	VAR robtarget OpenholeUD_6159 := [[399.17, -20.7, 180.93], [-0.152365, 0.690496, 0.688111, 0.1628], [0,0,0,0], [9E9, 9E9, 9E9, 9E9, 9E9, 9E9]];
	VAR robtarget OpenholeUD_6160 := [[395.17, -20.7, 180.87], [-0.163095, 0.688041, 0.685559, 0.173233], [0,0,0,0], [9E9, 9E9, 9E9, 9E9, 9E9, 9E9]];
	VAR robtarget OpenholeUD_6161 := [[389.34, -20.7, 180.77], [-0.17806, 0.684321, 0.681719, 0.187774], [0,0,0,0], [9E9, 9E9, 9E9, 9E9, 9E9, 9E9]];
	VAR robtarget OpenholeUD_6162 := [[385.34, -20.7, 180.79], [-0.183051, 0.683002, 0.683002, 0.183051], [0,0,0,0], [9E9, 9E9, 9E9, 9E9, 9E9, 9E9]];
	VAR robtarget OpenholeUD_6163 := [[381.34, -20.7, 180.8], [-0.183051, 0.683002, 0.683002, 0.183051], [0,0,0,0], [9E9, 9E9, 9E9, 9E9, 9E9, 9E9]];
	VAR robtarget OpenholeUD_6164 := [[377.34, -20.7, 180.81], [-0.183051, 0.683002, 0.683002, 0.183051], [0,0,0,0], [9E9, 9E9, 9E9, 9E9, 9E9, 9E9]];
	VAR robtarget OpenholeUD_6165 := [[373.34, -20.7, 180.83], [-0.183051, 0.683002, 0.683002, 0.183051], [0,0,0,0], [9E9, 9E9, 9E9, 9E9, 9E9, 9E9]];
	VAR robtarget OpenholeUD_6166 := [[369.34, -20.7, 180.84], [-0.183051, 0.683002, 0.683002, 0.183051], [0,0,0,0], [9E9, 9E9, 9E9, 9E9, 9E9, 9E9]];
	VAR robtarget OpenholeUD_6167 := [[369.34, -20.7, 180.84], [-0.183051, 0.683002, 0.683002, 0.183051], [0,0,0,0], [9E9, 9E9, 9E9, 9E9, 9E9, 9E9]];
	VAR robtarget OpenholeUD_6168 := [[369.35, -19.5, 181.53], [-0.183051, 0.683002, 0.683002, 0.183051], [0,0,0,0], [9E9, 9E9, 9E9, 9E9, 9E9, 9E9]];
	VAR robtarget OpenholeUD_6169 := [[373.35, -19.5, 181.52], [-0.183051, 0.683002, 0.683002, 0.183051], [0,0,0,0], [9E9, 9E9, 9E9, 9E9, 9E9, 9E9]];
	VAR robtarget OpenholeUD_6170 := [[377.35, -19.5, 181.51], [-0.183051, 0.683002, 0.683002, 0.183051], [0,0,0,0], [9E9, 9E9, 9E9, 9E9, 9E9, 9E9]];
	VAR robtarget OpenholeUD_6171 := [[381.35, -19.5, 181.49], [-0.183051, 0.683002, 0.683002, 0.183051], [0,0,0,0], [9E9, 9E9, 9E9, 9E9, 9E9, 9E9]];
	VAR robtarget OpenholeUD_6172 := [[385.35, -19.5, 181.48], [-0.183051, 0.683002, 0.683002, 0.183051], [0,0,0,0], [9E9, 9E9, 9E9, 9E9, 9E9, 9E9]];
	VAR robtarget OpenholeUD_6173 := [[389.35, -19.5, 181.47], [-0.18149, 0.683419, 0.682647, 0.18437], [0,0,0,0], [9E9, 9E9, 9E9, 9E9, 9E9, 9E9]];
	VAR robtarget OpenholeUD_6174 := [[393.35, -19.5, 181.49], [-0.171367, 0.686027, 0.685263, 0.174397], [0,0,0,0], [9E9, 9E9, 9E9, 9E9, 9E9, 9E9]];
	VAR robtarget OpenholeUD_6175 := [[397.35, -19.5, 181.5], [-0.160873, 0.688564, 0.687811, 0.164061], [0,0,0,0], [9E9, 9E9, 9E9, 9E9, 9E9, 9E9]];
	VAR robtarget OpenholeUD_6176 := [[401.35, -19.5, 181.52], [-0.15001, 0.691012, 0.690275, 0.153365], [0,0,0,0], [9E9, 9E9, 9E9, 9E9, 9E9, 9E9]];
	VAR robtarget OpenholeUD_6177 := [[405.35, -19.5, 181.54], [-0.138785, 0.693353, 0.692638, 0.142312], [0,0,0,0], [9E9, 9E9, 9E9, 9E9, 9E9, 9E9]];
	VAR robtarget OpenholeUD_6178 := [[409.35, -19.5, 181.56], [-0.127207, 0.695571, 0.694883, 0.130913], [0,0,0,0], [9E9, 9E9, 9E9, 9E9, 9E9, 9E9]];
	VAR robtarget OpenholeUD_6179 := [[413.35, -19.5, 181.58], [-0.11529, 0.697645, 0.696991, 0.11918], [0,0,0,0], [9E9, 9E9, 9E9, 9E9, 9E9, 9E9]];
	VAR robtarget OpenholeUD_6180 := [[417.35, -19.5, 181.6], [-0.103051, 0.699557, 0.698945, 0.107128], [0,0,0,0], [9E9, 9E9, 9E9, 9E9, 9E9, 9E9]];
	VAR robtarget OpenholeUD_6181 := [[421.35, -19.5, 181.61], [-0.090514, 0.70129, 0.700726, 0.09478], [0,0,0,0], [9E9, 9E9, 9E9, 9E9, 9E9, 9E9]];
	VAR robtarget OpenholeUD_6182 := [[425.35, -19.5, 181.63], [-0.077704, 0.702824, 0.702318, 0.082159], [0,0,0,0], [9E9, 9E9, 9E9, 9E9, 9E9, 9E9]];
	VAR robtarget OpenholeUD_6183 := [[429.35, -19.5, 181.65], [-0.064653, 0.704145, 0.703703, 0.069293], [0,0,0,0], [9E9, 9E9, 9E9, 9E9, 9E9, 9E9]];
	VAR robtarget OpenholeUD_6184 := [[433.35, -19.5, 181.67], [-0.051395, 0.705237, 0.704869, 0.056216], [0,0,0,0], [9E9, 9E9, 9E9, 9E9, 9E9, 9E9]];
	VAR robtarget OpenholeUD_6185 := [[437.35, -19.5, 181.69], [-0.037969, 0.706087, 0.7058, 0.042964], [0,0,0,0], [9E9, 9E9, 9E9, 9E9, 9E9, 9E9]];
	VAR robtarget OpenholeUD_6186 := [[442.9, -19.5, 181.71], [-0.019136, 0.706848, 0.706687, 0.024355], [0,0,0,0], [9E9, 9E9, 9E9, 9E9, 9E9, 9E9]];
	VAR robtarget OpenholeUD_6187 := [[442.9, -19.5, 181.71], [-0.019136, 0.706848, 0.706687, 0.024355], [0,0,0,0], [9E9, 9E9, 9E9, 9E9, 9E9, 9E9]];
	VAR robtarget OpenholeUD_6188 := [[442.86, -18.3, 181.79], [-0.023356, 0.706721, 0.706812, 0.020425], [0,0,0,0], [9E9, 9E9, 9E9, 9E9, 9E9, 9E9]];
	VAR robtarget OpenholeUD_6189 := [[438.86, -18.3, 181.81], [-0.03693, 0.706142, 0.706295, 0.033871], [0,0,0,0], [9E9, 9E9, 9E9, 9E9, 9E9, 9E9]];
	VAR robtarget OpenholeUD_6190 := [[434.86, -18.3, 181.84], [-0.050386, 0.705309, 0.705529, 0.047203], [0,0,0,0], [9E9, 9E9, 9E9, 9E9, 9E9, 9E9]];
	VAR robtarget OpenholeUD_6191 := [[430.86, -18.3, 181.87], [-0.063682, 0.704233, 0.704524, 0.06038], [0,0,0,0], [9E9, 9E9, 9E9, 9E9, 9E9, 9E9]];
	VAR robtarget OpenholeUD_6192 := [[426.86, -18.3, 181.9], [-0.076779, 0.702926, 0.70329, 0.073366], [0,0,0,0], [9E9, 9E9, 9E9, 9E9, 9E9, 9E9]];
	VAR robtarget OpenholeUD_6193 := [[422.86, -18.3, 181.93], [-0.089642, 0.701402, 0.701842, 0.086125], [0,0,0,0], [9E9, 9E9, 9E9, 9E9, 9E9, 9E9]];
	VAR robtarget OpenholeUD_6194 := [[418.86, -18.3, 181.95], [-0.102237, 0.699677, 0.700195, 0.098627], [0,0,0,0], [9E9, 9E9, 9E9, 9E9, 9E9, 9E9]];
	VAR robtarget OpenholeUD_6195 := [[414.86, -18.3, 181.98], [-0.114539, 0.697769, 0.698365, 0.110845], [0,0,0,0], [9E9, 9E9, 9E9, 9E9, 9E9, 9E9]];
	VAR robtarget OpenholeUD_6196 := [[410.86, -18.3, 182.01], [-0.126522, 0.695695, 0.69637, 0.122757], [0,0,0,0], [9E9, 9E9, 9E9, 9E9, 9E9, 9E9]];
	VAR robtarget OpenholeUD_6197 := [[406.86, -18.3, 182.04], [-0.138169, 0.693476, 0.694227, 0.134344], [0,0,0,0], [9E9, 9E9, 9E9, 9E9, 9E9, 9E9]];
	VAR robtarget OpenholeUD_6198 := [[402.86, -18.3, 182.07], [-0.149465, 0.69113, 0.691956, 0.145591], [0,0,0,0], [9E9, 9E9, 9E9, 9E9, 9E9, 9E9]];
	VAR robtarget OpenholeUD_6199 := [[398.86, -18.3, 182.09], [-0.160399, 0.688674, 0.689573, 0.156488], [0,0,0,0], [9E9, 9E9, 9E9, 9E9, 9E9, 9E9]];
	VAR robtarget OpenholeUD_6200 := [[394.86, -18.3, 182.12], [-0.170965, 0.686128, 0.687096, 0.167028], [0,0,0,0], [9E9, 9E9, 9E9, 9E9, 9E9, 9E9]];
	VAR robtarget OpenholeUD_6201 := [[389.35, -18.3, 182.16], [-0.184916, 0.6825, 0.683559, 0.180962], [0,0,0,0], [9E9, 9E9, 9E9, 9E9, 9E9, 9E9]];
	VAR robtarget OpenholeUD_6202 := [[385.35, -18.3, 182.17], [-0.183051, 0.683002, 0.683002, 0.183051], [0,0,0,0], [9E9, 9E9, 9E9, 9E9, 9E9, 9E9]];
	VAR robtarget OpenholeUD_6203 := [[381.35, -18.3, 182.19], [-0.183051, 0.683002, 0.683002, 0.183051], [0,0,0,0], [9E9, 9E9, 9E9, 9E9, 9E9, 9E9]];
	VAR robtarget OpenholeUD_6204 := [[377.35, -18.3, 182.2], [-0.183051, 0.683002, 0.683002, 0.183051], [0,0,0,0], [9E9, 9E9, 9E9, 9E9, 9E9, 9E9]];
	VAR robtarget OpenholeUD_6205 := [[373.35, -18.3, 182.21], [-0.183051, 0.683002, 0.683002, 0.183051], [0,0,0,0], [9E9, 9E9, 9E9, 9E9, 9E9, 9E9]];
	VAR robtarget OpenholeUD_6206 := [[369.35, -18.3, 182.22], [-0.183051, 0.683002, 0.683002, 0.183051], [0,0,0,0], [9E9, 9E9, 9E9, 9E9, 9E9, 9E9]];
	VAR robtarget OpenholeUD_6207 := [[369.35, -18.3, 182.22], [-0.183051, 0.683002, 0.683002, 0.183051], [0,0,0,0], [9E9, 9E9, 9E9, 9E9, 9E9, 9E9]];
	VAR robtarget OpenholeUD_6208 := [[369.35, -17.1, 182.92], [-0.183051, 0.683002, 0.683002, 0.183051], [0,0,0,0], [9E9, 9E9, 9E9, 9E9, 9E9, 9E9]];
	VAR robtarget OpenholeUD_6209 := [[373.35, -17.1, 182.9], [-0.183051, 0.683002, 0.683002, 0.183051], [0,0,0,0], [9E9, 9E9, 9E9, 9E9, 9E9, 9E9]];
	VAR robtarget OpenholeUD_6210 := [[377.35, -17.1, 182.89], [-0.183051, 0.683002, 0.683002, 0.183051], [0,0,0,0], [9E9, 9E9, 9E9, 9E9, 9E9, 9E9]];
	VAR robtarget OpenholeUD_6211 := [[381.35, -17.1, 182.88], [-0.183051, 0.683002, 0.683002, 0.183051], [0,0,0,0], [9E9, 9E9, 9E9, 9E9, 9E9, 9E9]];
	VAR robtarget OpenholeUD_6212 := [[389.35, -17.1, 182.85], [-0.188337, 0.681564, 0.684453, 0.17755], [0,0,0,0], [9E9, 9E9, 9E9, 9E9, 9E9, 9E9]];
	VAR robtarget OpenholeUD_6213 := [[393.35, -17.1, 182.78], [-0.178356, 0.684243, 0.686996, 0.167441], [0,0,0,0], [9E9, 9E9, 9E9, 9E9, 9E9, 9E9]];
	VAR robtarget OpenholeUD_6214 := [[397.35, -17.1, 182.71], [-0.168002, 0.686859, 0.689464, 0.156971], [0,0,0,0], [9E9, 9E9, 9E9, 9E9, 9E9, 9E9]];
	VAR robtarget OpenholeUD_6215 := [[401.35, -17.1, 182.63], [-0.157276, 0.689394, 0.69184, 0.146144], [0,0,0,0], [9E9, 9E9, 9E9, 9E9, 9E9, 9E9]];
	VAR robtarget OpenholeUD_6216 := [[405.35, -17.1, 182.56], [-0.146183, 0.691831, 0.694107, 0.134966], [0,0,0,0], [9E9, 9E9, 9E9, 9E9, 9E9, 9E9]];
	VAR robtarget OpenholeUD_6217 := [[409.35, -17.1, 182.48], [-0.134731, 0.694152, 0.696248, 0.123447], [0,0,0,0], [9E9, 9E9, 9E9, 9E9, 9E9, 9E9]];
	VAR robtarget OpenholeUD_6218 := [[413.35, -17.1, 182.41], [-0.122934, 0.696338, 0.698244, 0.111601], [0,0,0,0], [9E9, 9E9, 9E9, 9E9, 9E9, 9E9]];
	VAR robtarget OpenholeUD_6219 := [[417.35, -17.1, 182.33], [-0.110807, 0.698371, 0.700079, 0.099445], [0,0,0,0], [9E9, 9E9, 9E9, 9E9, 9E9, 9E9]];
	VAR robtarget OpenholeUD_6220 := [[421.35, -17.1, 182.26], [-0.098372, 0.700231, 0.701734, 0.087], [0,0,0,0], [9E9, 9E9, 9E9, 9E9, 9E9, 9E9]];
	VAR robtarget OpenholeUD_6221 := [[425.34, -17.1, 182.19], [-0.085654, 0.7019, 0.703193, 0.074294], [0,0,0,0], [9E9, 9E9, 9E9, 9E9, 9E9, 9E9]];
	VAR robtarget OpenholeUD_6222 := [[429.34, -17.1, 182.11], [-0.072683, 0.703361, 0.70444, 0.061354], [0,0,0,0], [9E9, 9E9, 9E9, 9E9, 9E9, 9E9]];
	VAR robtarget OpenholeUD_6223 := [[433.34, -17.1, 182.04], [-0.059492, 0.7046, 0.705461, 0.048215], [0,0,0,0], [9E9, 9E9, 9E9, 9E9, 9E9, 9E9]];
	VAR robtarget OpenholeUD_6224 := [[437.34, -17.1, 181.96], [-0.04612, 0.705601, 0.706244, 0.034914], [0,0,0,0], [9E9, 9E9, 9E9, 9E9, 9E9, 9E9]];
	VAR robtarget OpenholeUD_6225 := [[443.05, -17.1, 181.86], [-0.02681, 0.706598, 0.706932, 0.015737], [0,0,0,0], [9E9, 9E9, 9E9, 9E9, 9E9, 9E9]];
	VAR robtarget OpenholeUD_6226 := [[443.05, -17.1, 181.86], [-0.02681, 0.706598, 0.706932, 0.015737], [0,0,0,0], [9E9, 9E9, 9E9, 9E9, 9E9, 9E9]];
	VAR robtarget OpenholeUD_6227 := [[443.48, -15.9, 181.92], [-0.029424, 0.706494, 0.707033, 0.010217], [0,0,0,0], [9E9, 9E9, 9E9, 9E9, 9E9, 9E9]];
	VAR robtarget OpenholeUD_6228 := [[439.48, -15.9, 182.04], [-0.042977, 0.7058, 0.70671, 0.023699], [0,0,0,0], [9E9, 9E9, 9E9, 9E9, 9E9, 9E9]];
	VAR robtarget OpenholeUD_6229 := [[435.49, -15.9, 182.16], [-0.056403, 0.704854, 0.706133, 0.037088], [0,0,0,0], [9E9, 9E9, 9E9, 9E9, 9E9, 9E9]];
	VAR robtarget OpenholeUD_6230 := [[431.49, -15.9, 182.28], [-0.069663, 0.703667, 0.705312, 0.050343], [0,0,0,0], [9E9, 9E9, 9E9, 9E9, 9E9, 9E9]];
	VAR robtarget OpenholeUD_6231 := [[427.49, -15.9, 182.4], [-0.082716, 0.702252, 0.704257, 0.063424], [0,0,0,0], [9E9, 9E9, 9E9, 9E9, 9E9, 9E9]];
	VAR robtarget OpenholeUD_6232 := [[423.49, -15.9, 182.52], [-0.095528, 0.700624, 0.702979, 0.076296], [0,0,0,0], [9E9, 9E9, 9E9, 9E9, 9E9, 9E9]];
	VAR robtarget OpenholeUD_6233 := [[419.49, -15.9, 182.64], [-0.108067, 0.6988, 0.701493, 0.088927], [0,0,0,0], [9E9, 9E9, 9E9, 9E9, 9E9, 9E9]];
	VAR robtarget OpenholeUD_6234 := [[415.49, -15.9, 182.76], [-0.120306, 0.696797, 0.699815, 0.101288], [0,0,0,0], [9E9, 9E9, 9E9, 9E9, 9E9, 9E9]];
	VAR robtarget OpenholeUD_6235 := [[411.5, -15.9, 182.88], [-0.132222, 0.694635, 0.697962, 0.113355], [0,0,0,0], [9E9, 9E9, 9E9, 9E9, 9E9, 9E9]];
	VAR robtarget OpenholeUD_6236 := [[407.5, -15.9, 183], [-0.143797, 0.692331, 0.695951, 0.125107], [0,0,0,0], [9E9, 9E9, 9E9, 9E9, 9E9, 9E9]];
	VAR robtarget OpenholeUD_6237 := [[403.5, -15.9, 183.12], [-0.155017, 0.689906, 0.693801, 0.136528], [0,0,0,0], [9E9, 9E9, 9E9, 9E9, 9E9, 9E9]];
	VAR robtarget OpenholeUD_6238 := [[399.5, -15.9, 183.24], [-0.165872, 0.687377, 0.691529, 0.147606], [0,0,0,0], [9E9, 9E9, 9E9, 9E9, 9E9, 9E9]];
	VAR robtarget OpenholeUD_6239 := [[395.5, -15.9, 183.36], [-0.176355, 0.684762, 0.689152, 0.158332], [0,0,0,0], [9E9, 9E9, 9E9, 9E9, 9E9, 9E9]];
	VAR robtarget OpenholeUD_6240 := [[389.35, -15.9, 183.55], [-0.191751, 0.680611, 0.68533, 0.174134], [0,0,0,0], [9E9, 9E9, 9E9, 9E9, 9E9, 9E9]];
	VAR robtarget OpenholeUD_6241 := [[385.35, -15.9, 183.56], [-0.183051, 0.683002, 0.683002, 0.183051], [0,0,0,0], [9E9, 9E9, 9E9, 9E9, 9E9, 9E9]];
	VAR robtarget OpenholeUD_6242 := [[381.35, -15.9, 183.57], [-0.183051, 0.683002, 0.683002, 0.183051], [0,0,0,0], [9E9, 9E9, 9E9, 9E9, 9E9, 9E9]];
	VAR robtarget OpenholeUD_6243 := [[377.35, -15.9, 183.58], [-0.183051, 0.683002, 0.683002, 0.183051], [0,0,0,0], [9E9, 9E9, 9E9, 9E9, 9E9, 9E9]];
	VAR robtarget OpenholeUD_6244 := [[369.35, -15.9, 183.61], [-0.183051, 0.683002, 0.683002, 0.183051], [0,0,0,0], [9E9, 9E9, 9E9, 9E9, 9E9, 9E9]];
	VAR robtarget OpenholeUD_6245 := [[369.35, -15.9, 183.61], [-0.183051, 0.683002, 0.683002, 0.183051], [0,0,0,0], [9E9, 9E9, 9E9, 9E9, 9E9, 9E9]];
	VAR robtarget OpenholeUD_6246 := [[369.36, -14.7, 184.3], [-0.183051, 0.683002, 0.683002, 0.183051], [0,0,0,0], [9E9, 9E9, 9E9, 9E9, 9E9, 9E9]];
	VAR robtarget OpenholeUD_6247 := [[373.36, -14.7, 184.29], [-0.183051, 0.683002, 0.683002, 0.183051], [0,0,0,0], [9E9, 9E9, 9E9, 9E9, 9E9, 9E9]];
	VAR robtarget OpenholeUD_6248 := [[377.36, -14.7, 184.28], [-0.183051, 0.683002, 0.683002, 0.183051], [0,0,0,0], [9E9, 9E9, 9E9, 9E9, 9E9, 9E9]];
	VAR robtarget OpenholeUD_6249 := [[381.36, -14.7, 184.27], [-0.183051, 0.683002, 0.683002, 0.183051], [0,0,0,0], [9E9, 9E9, 9E9, 9E9, 9E9, 9E9]];
	VAR robtarget OpenholeUD_6250 := [[389.36, -14.7, 184.24], [-0.195159, 0.679642, 0.686189, 0.170717], [0,0,0,0], [9E9, 9E9, 9E9, 9E9, 9E9, 9E9]];
	VAR robtarget OpenholeUD_6251 := [[393.35, -14.7, 184.07], [-0.185327, 0.682389, 0.688656, 0.160477], [0,0,0,0], [9E9, 9E9, 9E9, 9E9, 9E9, 9E9]];
	VAR robtarget OpenholeUD_6252 := [[397.35, -14.7, 183.91], [-0.175118, 0.685079, 0.69104, 0.149881], [0,0,0,0], [9E9, 9E9, 9E9, 9E9, 9E9, 9E9]];
	VAR robtarget OpenholeUD_6253 := [[401.34, -14.7, 183.74], [-0.164535, 0.687698, 0.693324, 0.138931], [0,0,0,0], [9E9, 9E9, 9E9, 9E9, 9E9, 9E9]];
	VAR robtarget OpenholeUD_6254 := [[405.34, -14.7, 183.57], [-0.153582, 0.690227, 0.695492, 0.127635], [0,0,0,0], [9E9, 9E9, 9E9, 9E9, 9E9, 9E9]];
	VAR robtarget OpenholeUD_6255 := [[409.34, -14.7, 183.41], [-0.142264, 0.692648, 0.697526, 0.116004], [0,0,0,0], [9E9, 9E9, 9E9, 9E9, 9E9, 9E9]];
	VAR robtarget OpenholeUD_6256 := [[413.33, -14.7, 183.24], [-0.130595, 0.694942, 0.699409, 0.104054], [0,0,0,0], [9E9, 9E9, 9E9, 9E9, 9E9, 9E9]];
	VAR robtarget OpenholeUD_6257 := [[417.33, -14.7, 183.07], [-0.118588, 0.697092, 0.701122, 0.091801], [0,0,0,0], [9E9, 9E9, 9E9, 9E9, 9E9, 9E9]];
	VAR robtarget OpenholeUD_6258 := [[421.33, -14.7, 182.91], [-0.106265, 0.699076, 0.702649, 0.079271], [0,0,0,0], [9E9, 9E9, 9E9, 9E9, 9E9, 9E9]];
	VAR robtarget OpenholeUD_6259 := [[425.32, -14.7, 182.74], [-0.093648, 0.700878, 0.703974, 0.066488], [0,0,0,0], [9E9, 9E9, 9E9, 9E9, 9E9, 9E9]];
	VAR robtarget OpenholeUD_6260 := [[429.32, -14.7, 182.58], [-0.080766, 0.702479, 0.705081, 0.053484], [0,0,0,0], [9E9, 9E9, 9E9, 9E9, 9E9, 9E9]];
	VAR robtarget OpenholeUD_6261 := [[433.32, -14.7, 182.41], [-0.067653, 0.703863, 0.705958, 0.040293], [0,0,0,0], [9E9, 9E9, 9E9, 9E9, 9E9, 9E9]];
	VAR robtarget OpenholeUD_6262 := [[437.31, -14.7, 182.24], [-0.054344, 0.705015, 0.706593, 0.026953], [0,0,0,0], [9E9, 9E9, 9E9, 9E9, 9E9, 9E9]];
	VAR robtarget OpenholeUD_6263 := [[444.22, -14.7, 181.95], [-0.030987, 0.706427, 0.707097, 0.003651], [0,0,0,0], [9E9, 9E9, 9E9, 9E9, 9E9, 9E9]];
	VAR robtarget OpenholeUD_6264 := [[444.22, -14.7, 181.95], [-0.030987, 0.706427, 0.707097, 0.003651], [0,0,0,0], [9E9, 9E9, 9E9, 9E9, 9E9, 9E9]];
	VAR robtarget OpenholeUD_6265 := [[445.45, -13.5, 181.95], [-0.030912, 0.706431, 0.707092, -0.004543], [0,0,0,0], [9E9, 9E9, 9E9, 9E9, 9E9, 9E9]];
	VAR robtarget OpenholeUD_6266 := [[441.45, -13.5, 182.16], [-0.044472, 0.705707, 0.70705, 0.008977], [0,0,0,0], [9E9, 9E9, 9E9, 9E9, 9E9, 9E9]];
	VAR robtarget OpenholeUD_6267 := [[437.46, -13.5, 182.37], [-0.057913, 0.704731, 0.706751, 0.022438], [0,0,0,0], [9E9, 9E9, 9E9, 9E9, 9E9, 9E9]];
	VAR robtarget OpenholeUD_6268 := [[433.46, -13.5, 182.59], [-0.071194, 0.703514, 0.7062, 0.0358], [0,0,0,0], [9E9, 9E9, 9E9, 9E9, 9E9, 9E9]];
	VAR robtarget OpenholeUD_6269 := [[429.47, -13.5, 182.8], [-0.084275, 0.702067, 0.705406, 0.04902], [0,0,0,0], [9E9, 9E9, 9E9, 9E9, 9E9, 9E9]];
	VAR robtarget OpenholeUD_6270 := [[425.48, -13.5, 183.01], [-0.097118, 0.700406, 0.704378, 0.062061], [0,0,0,0], [9E9, 9E9, 9E9, 9E9, 9E9, 9E9]];
	VAR robtarget OpenholeUD_6271 := [[421.48, -13.5, 183.22], [-0.109693, 0.698547, 0.70313, 0.074888], [0,0,0,0], [9E9, 9E9, 9E9, 9E9, 9E9, 9E9]];
	VAR robtarget OpenholeUD_6272 := [[417.49, -13.5, 183.44], [-0.121971, 0.696508, 0.701676, 0.08747], [0,0,0,0], [9E9, 9E9, 9E9, 9E9, 9E9, 9E9]];
	VAR robtarget OpenholeUD_6273 := [[413.49, -13.5, 183.65], [-0.133929, 0.694308, 0.700032, 0.099779], [0,0,0,0], [9E9, 9E9, 9E9, 9E9, 9E9, 9E9]];
	VAR robtarget OpenholeUD_6274 := [[409.5, -13.5, 183.86], [-0.145546, 0.691966, 0.698214, 0.111792], [0,0,0,0], [9E9, 9E9, 9E9, 9E9, 9E9, 9E9]];
	VAR robtarget OpenholeUD_6275 := [[405.5, -13.5, 184.07], [-0.156809, 0.6895, 0.69624, 0.123489], [0,0,0,0], [9E9, 9E9, 9E9, 9E9, 9E9, 9E9]];
	VAR robtarget OpenholeUD_6276 := [[401.51, -13.5, 184.29], [-0.167706, 0.686931, 0.694128, 0.134855], [0,0,0,0], [9E9, 9E9, 9E9, 9E9, 9E9, 9E9]];
	VAR robtarget OpenholeUD_6277 := [[397.52, -13.5, 184.5], [-0.178231, 0.684276, 0.691896, 0.145878], [0,0,0,0], [9E9, 9E9, 9E9, 9E9, 9E9, 9E9]];
	VAR robtarget OpenholeUD_6278 := [[393.52, -13.5, 184.71], [-0.18838, 0.681552, 0.689559, 0.156551], [0,0,0,0], [9E9, 9E9, 9E9, 9E9, 9E9, 9E9]];
	VAR robtarget OpenholeUD_6279 := [[389.36, -13.5, 184.93], [-0.19856, 0.678656, 0.687031, 0.167297], [0,0,0,0], [9E9, 9E9, 9E9, 9E9, 9E9, 9E9]];
	VAR robtarget OpenholeUD_6280 := [[385.36, -13.5, 184.95], [-0.183051, 0.683002, 0.683002, 0.183051], [0,0,0,0], [9E9, 9E9, 9E9, 9E9, 9E9, 9E9]];
	VAR robtarget OpenholeUD_6281 := [[381.36, -13.5, 184.96], [-0.183051, 0.683002, 0.683002, 0.183051], [0,0,0,0], [9E9, 9E9, 9E9, 9E9, 9E9, 9E9]];
	VAR robtarget OpenholeUD_6282 := [[377.36, -13.5, 184.97], [-0.183051, 0.683002, 0.683002, 0.183051], [0,0,0,0], [9E9, 9E9, 9E9, 9E9, 9E9, 9E9]];
	VAR robtarget OpenholeUD_6283 := [[369.36, -13.5, 185], [-0.183051, 0.683002, 0.683002, 0.183051], [0,0,0,0], [9E9, 9E9, 9E9, 9E9, 9E9, 9E9]];
	VAR robtarget OpenholeUD_6284 := [[369.36, -13.5, 185], [-0.183051, 0.683002, 0.683002, 0.183051], [0,0,0,0], [9E9, 9E9, 9E9, 9E9, 9E9, 9E9]];
	VAR robtarget OpenholeUD_6285 := [[369.36, -12.3, 185.69], [-0.183051, 0.683002, 0.683002, 0.183051], [0,0,0,0], [9E9, 9E9, 9E9, 9E9, 9E9, 9E9]];
	VAR robtarget OpenholeUD_6286 := [[373.36, -12.3, 185.68], [-0.183051, 0.683002, 0.683002, 0.183051], [0,0,0,0], [9E9, 9E9, 9E9, 9E9, 9E9, 9E9]];
	VAR robtarget OpenholeUD_6287 := [[377.36, -12.3, 185.66], [-0.183051, 0.683002, 0.683002, 0.183051], [0,0,0,0], [9E9, 9E9, 9E9, 9E9, 9E9, 9E9]];
	VAR robtarget OpenholeUD_6288 := [[381.36, -12.3, 185.65], [-0.183051, 0.683002, 0.683002, 0.183051], [0,0,0,0], [9E9, 9E9, 9E9, 9E9, 9E9, 9E9]];
	VAR robtarget OpenholeUD_6289 := [[385.36, -12.3, 185.64], [-0.183051, 0.683002, 0.683002, 0.183051], [0,0,0,0], [9E9, 9E9, 9E9, 9E9, 9E9, 9E9]];
	VAR robtarget OpenholeUD_6290 := [[389.36, -12.3, 185.63], [-0.201952, 0.677654, 0.687855, 0.163877], [0,0,0,0], [9E9, 9E9, 9E9, 9E9, 9E9, 9E9]];
	VAR robtarget OpenholeUD_6291 := [[393.35, -12.3, 185.37], [-0.192272, 0.680464, 0.690241, 0.153515], [0,0,0,0], [9E9, 9E9, 9E9, 9E9, 9E9, 9E9]];
	VAR robtarget OpenholeUD_6292 := [[397.34, -12.3, 185.11], [-0.182215, 0.683226, 0.692538, 0.142798], [0,0,0,0], [9E9, 9E9, 9E9, 9E9, 9E9, 9E9]];
	VAR robtarget OpenholeUD_6293 := [[401.33, -12.3, 184.85], [-0.171781, 0.685924, 0.694728, 0.131733], [0,0,0,0], [9E9, 9E9, 9E9, 9E9, 9E9, 9E9]];
	VAR robtarget OpenholeUD_6294 := [[405.33, -12.3, 184.59], [-0.160973, 0.68854, 0.696794, 0.120328], [0,0,0,0], [9E9, 9E9, 9E9, 9E9, 9E9, 9E9]];
	VAR robtarget OpenholeUD_6295 := [[409.32, -12.3, 184.33], [-0.149797, 0.691058, 0.698718, 0.108594], [0,0,0,0], [9E9, 9E9, 9E9, 9E9, 9E9, 9E9]];
	VAR robtarget OpenholeUD_6296 := [[413.31, -12.3, 184.08], [-0.138263, 0.693458, 0.700485, 0.096548], [0,0,0,0], [9E9, 9E9, 9E9, 9E9, 9E9, 9E9]];
	VAR robtarget OpenholeUD_6297 := [[417.3, -12.3, 183.82], [-0.126385, 0.69572, 0.702075, 0.084208], [0,0,0,0], [9E9, 9E9, 9E9, 9E9, 9E9, 9E9]];
	VAR robtarget OpenholeUD_6298 := [[421.29, -12.3, 183.56], [-0.114181, 0.697827, 0.703472, 0.0716], [0,0,0,0], [9E9, 9E9, 9E9, 9E9, 9E9, 9E9]];
	VAR robtarget OpenholeUD_6299 := [[425.28, -12.3, 183.3], [-0.101674, 0.699759, 0.704662, 0.058751], [0,0,0,0], [9E9, 9E9, 9E9, 9E9, 9E9, 9E9]];
	VAR robtarget OpenholeUD_6300 := [[429.28, -12.3, 183.04], [-0.088892, 0.701497, 0.705629, 0.045692], [0,0,0,0], [9E9, 9E9, 9E9, 9E9, 9E9, 9E9]];
	VAR robtarget OpenholeUD_6301 := [[433.27, -12.3, 182.78], [-0.075866, 0.703025, 0.706361, 0.032458], [0,0,0,0], [9E9, 9E9, 9E9, 9E9, 9E9, 9E9]];
	VAR robtarget OpenholeUD_6302 := [[437.26, -12.3, 182.52], [-0.062631, 0.704328, 0.706849, 0.019088], [0,0,0,0], [9E9, 9E9, 9E9, 9E9, 9E9, 9E9]];
	VAR robtarget OpenholeUD_6303 := [[441.25, -12.3, 182.27], [-0.049226, 0.705391, 0.707084, 0.005623], [0,0,0,0], [9E9, 9E9, 9E9, 9E9, 9E9, 9E9]];
	VAR robtarget OpenholeUD_6304 := [[445.24, -12.3, 182.01], [-0.035693, 0.706205, 0.707063, -0.007895], [0,0,0,0], [9E9, 9E9, 9E9, 9E9, 9E9, 9E9]];
	VAR robtarget OpenholeUD_6305 := [[449.23, -12.3, 181.75], [-0.022077, 0.706762, 0.706782, -0.021422], [0,0,0,0], [9E9, 9E9, 9E9, 9E9, 9E9, 9E9]];
	VAR robtarget OpenholeUD_6306 := [[453.23, -12.3, 181.49], [-0.008423, 0.707057, 0.706244, -0.034914], [0,0,0,0], [9E9, 9E9, 9E9, 9E9, 9E9, 9E9]];
	VAR robtarget OpenholeUD_6307 := [[457.22, -12.3, 181.23], [0.005224, 0.707087, 0.705453, -0.048326], [0,0,0,0], [9E9, 9E9, 9E9, 9E9, 9E9, 9E9]];
	VAR robtarget OpenholeUD_6308 := [[461.21, -12.3, 180.97], [0.018817, 0.706856, 0.704417, -0.061617], [0,0,0,0], [9E9, 9E9, 9E9, 9E9, 9E9, 9E9]];
	VAR robtarget OpenholeUD_6309 := [[465.2, -12.3, 180.71], [0.032313, 0.706368, 0.703145, -0.074746], [0,0,0,0], [9E9, 9E9, 9E9, 9E9, 9E9, 9E9]];
	VAR robtarget OpenholeUD_6310 := [[469.19, -12.3, 180.46], [0.045667, 0.705631, 0.70165, -0.087675], [0,0,0,0], [9E9, 9E9, 9E9, 9E9, 9E9, 9E9]];
	VAR robtarget OpenholeUD_6311 := [[473.18, -12.3, 180.2], [0.058842, 0.704654, 0.699947, -0.10037], [0,0,0,0], [9E9, 9E9, 9E9, 9E9, 9E9, 9E9]];
	VAR robtarget OpenholeUD_6312 := [[477.18, -12.3, 179.94], [0.0718, 0.703452, 0.698052, -0.112799], [0,0,0,0], [9E9, 9E9, 9E9, 9E9, 9E9, 9E9]];
	VAR robtarget OpenholeUD_6313 := [[481.17, -12.3, 179.68], [0.08451, 0.702039, 0.695982, -0.124937], [0,0,0,0], [9E9, 9E9, 9E9, 9E9, 9E9, 9E9]];
	VAR robtarget OpenholeUD_6314 := [[485.16, -12.3, 179.42], [0.096942, 0.70043, 0.693756, -0.13676], [0,0,0,0], [9E9, 9E9, 9E9, 9E9, 9E9, 9E9]];
	VAR robtarget OpenholeUD_6315 := [[489.15, -12.3, 179.16], [0.109072, 0.698644, 0.691391, -0.148249], [0,0,0,0], [9E9, 9E9, 9E9, 9E9, 9E9, 9E9]];
	VAR robtarget OpenholeUD_6316 := [[493.14, -12.3, 178.91], [0.12088, 0.696698, 0.688908, -0.159391], [0,0,0,0], [9E9, 9E9, 9E9, 9E9, 9E9, 9E9]];
	VAR robtarget OpenholeUD_6317 := [[497.13, -12.3, 178.65], [0.132351, 0.69461, 0.686324, -0.170175], [0,0,0,0], [9E9, 9E9, 9E9, 9E9, 9E9, 9E9]];
	VAR robtarget OpenholeUD_6318 := [[501.13, -12.3, 178.39], [0.143473, 0.692398, 0.683656, -0.180593], [0,0,0,0], [9E9, 9E9, 9E9, 9E9, 9E9, 9E9]];
	VAR robtarget OpenholeUD_6319 := [[505.12, -12.3, 178.13], [0.154238, 0.69008, 0.680922, -0.190644], [0,0,0,0], [9E9, 9E9, 9E9, 9E9, 9E9, 9E9]];
	VAR robtarget OpenholeUD_6320 := [[509.34, -12.3, 177.86], [0.183051, 0.683002, 0.683002, -0.183051], [0,0,0,0], [9E9, 9E9, 9E9, 9E9, 9E9, 9E9]];
	VAR robtarget OpenholeUD_6321 := [[513.34, -12.3, 177.84], [0.183051, 0.683002, 0.683002, -0.183051], [0,0,0,0], [9E9, 9E9, 9E9, 9E9, 9E9, 9E9]];
	VAR robtarget OpenholeUD_6322 := [[517.34, -12.3, 177.83], [0.183051, 0.683002, 0.683002, -0.183051], [0,0,0,0], [9E9, 9E9, 9E9, 9E9, 9E9, 9E9]];
	VAR robtarget OpenholeUD_6323 := [[521.34, -12.3, 177.82], [0.183051, 0.683002, 0.683002, -0.183051], [0,0,0,0], [9E9, 9E9, 9E9, 9E9, 9E9, 9E9]];
	VAR robtarget OpenholeUD_6324 := [[529.34, -12.3, 177.79], [0.183051, 0.683002, 0.683002, -0.183051], [0,0,0,0], [9E9, 9E9, 9E9, 9E9, 9E9, 9E9]];
	VAR robtarget OpenholeUD_6325 := [[529.34, -12.3, 177.79], [0.183051, 0.683002, 0.683002, -0.183051], [0,0,0,0], [9E9, 9E9, 9E9, 9E9, 9E9, 9E9]];
	VAR robtarget OpenholeUD_6326 := [[529.34, -13.5, 178.49], [0.183051, 0.683002, 0.683002, -0.183051], [0,0,0,0], [9E9, 9E9, 9E9, 9E9, 9E9, 9E9]];
	VAR robtarget OpenholeUD_6327 := [[525.34, -13.5, 178.5], [0.183051, 0.683002, 0.683002, -0.183051], [0,0,0,0], [9E9, 9E9, 9E9, 9E9, 9E9, 9E9]];
	VAR robtarget OpenholeUD_6328 := [[521.34, -13.5, 178.51], [0.183051, 0.683002, 0.683002, -0.183051], [0,0,0,0], [9E9, 9E9, 9E9, 9E9, 9E9, 9E9]];
	VAR robtarget OpenholeUD_6329 := [[517.34, -13.5, 178.52], [0.183051, 0.683002, 0.683002, -0.183051], [0,0,0,0], [9E9, 9E9, 9E9, 9E9, 9E9, 9E9]];
	VAR robtarget OpenholeUD_6330 := [[513.34, -13.5, 178.54], [0.183051, 0.683002, 0.683002, -0.183051], [0,0,0,0], [9E9, 9E9, 9E9, 9E9, 9E9, 9E9]];
	VAR robtarget OpenholeUD_6331 := [[509.34, -13.5, 178.55], [0.183051, 0.683002, 0.683002, -0.183051], [0,0,0,0], [9E9, 9E9, 9E9, 9E9, 9E9, 9E9]];
	VAR robtarget OpenholeUD_6332 := [[505.34, -13.5, 178.76], [0.158342, 0.68915, 0.681724, -0.187755], [0,0,0,0], [9E9, 9E9, 9E9, 9E9, 9E9, 9E9]];
	VAR robtarget OpenholeUD_6333 := [[501.35, -13.5, 178.97], [0.147659, 0.691518, 0.684427, -0.177651], [0,0,0,0], [9E9, 9E9, 9E9, 9E9, 9E9, 9E9]];
	VAR robtarget OpenholeUD_6334 := [[497.35, -13.5, 179.19], [0.136615, 0.693784, 0.68706, -0.16718], [0,0,0,0], [9E9, 9E9, 9E9, 9E9, 9E9, 9E9]];
	VAR robtarget OpenholeUD_6335 := [[493.36, -13.5, 179.4], [0.125219, 0.695931, 0.689606, -0.156345], [0,0,0,0], [9E9, 9E9, 9E9, 9E9, 9E9, 9E9]];
	VAR robtarget OpenholeUD_6336 := [[489.37, -13.5, 179.61], [0.113482, 0.697941, 0.692048, -0.145153], [0,0,0,0], [9E9, 9E9, 9E9, 9E9, 9E9, 9E9]];
	VAR robtarget OpenholeUD_6337 := [[485.37, -13.5, 179.82], [0.101418, 0.699796, 0.694368, -0.133616], [0,0,0,0], [9E9, 9E9, 9E9, 9E9, 9E9, 9E9]];
	VAR robtarget OpenholeUD_6338 := [[481.38, -13.5, 180.04], [0.089046, 0.701478, 0.696547, -0.121748], [0,0,0,0], [9E9, 9E9, 9E9, 9E9, 9E9, 9E9]];
	VAR robtarget OpenholeUD_6339 := [[477.38, -13.5, 180.25], [0.076391, 0.702968, 0.698566, -0.109569], [0,0,0,0], [9E9, 9E9, 9E9, 9E9, 9E9, 9E9]];
	VAR robtarget OpenholeUD_6340 := [[473.39, -13.5, 180.46], [0.063479, 0.704252, 0.700408, -0.097101], [0,0,0,0], [9E9, 9E9, 9E9, 9E9, 9E9, 9E9]];
	VAR robtarget OpenholeUD_6341 := [[469.39, -13.5, 180.67], [0.050343, 0.705312, 0.702055, -0.084371], [0,0,0,0], [9E9, 9E9, 9E9, 9E9, 9E9, 9E9]];
	VAR robtarget OpenholeUD_6342 := [[465.4, -13.5, 180.89], [0.037018, 0.706137, 0.703492, -0.071411], [0,0,0,0], [9E9, 9E9, 9E9, 9E9, 9E9, 9E9]];
	VAR robtarget OpenholeUD_6343 := [[461.41, -13.5, 181.1], [0.023544, 0.706715, 0.704703, -0.058256], [0,0,0,0], [9E9, 9E9, 9E9, 9E9, 9E9, 9E9]];
	VAR robtarget OpenholeUD_6344 := [[457.41, -13.5, 181.31], [0.009963, 0.707037, 0.705677, -0.044943], [0,0,0,0], [9E9, 9E9, 9E9, 9E9, 9E9, 9E9]];
	VAR robtarget OpenholeUD_6345 := [[453.25, -13.5, 181.53], [-0.004261, 0.707094, 0.706429, -0.030942], [0,0,0,0], [9E9, 9E9, 9E9, 9E9, 9E9, 9E9]];
	VAR robtarget OpenholeUD_6346 := [[453.25, -13.5, 181.53], [-0.004261, 0.707094, 0.706429, -0.030942], [0,0,0,0], [9E9, 9E9, 9E9, 9E9, 9E9, 9E9]];
	VAR robtarget OpenholeUD_6347 := [[454.47, -14.7, 181.53], [0.00401, 0.707095, 0.706426, -0.031017], [0,0,0,0], [9E9, 9E9, 9E9, 9E9, 9E9, 9E9]];
	VAR robtarget OpenholeUD_6348 := [[458.47, -14.7, 181.36], [0.017638, 0.706887, 0.705709, -0.044441], [0,0,0,0], [9E9, 9E9, 9E9, 9E9, 9E9, 9E9]];
	VAR robtarget OpenholeUD_6349 := [[462.46, -14.7, 181.2], [0.031183, 0.706419, 0.704745, -0.057745], [0,0,0,0], [9E9, 9E9, 9E9, 9E9, 9E9, 9E9]];
	VAR robtarget OpenholeUD_6350 := [[466.46, -14.7, 181.03], [0.044602, 0.705699, 0.703545, -0.070887], [0,0,0,0], [9E9, 9E9, 9E9, 9E9, 9E9, 9E9]];
	VAR robtarget OpenholeUD_6351 := [[470.46, -14.7, 180.86], [0.057854, 0.704736, 0.70212, -0.083831], [0,0,0,0], [9E9, 9E9, 9E9, 9E9, 9E9, 9E9]];
	VAR robtarget OpenholeUD_6352 := [[474.45, -14.7, 180.7], [0.070901, 0.703543, 0.700485, -0.096541], [0,0,0,0], [9E9, 9E9, 9E9, 9E9, 9E9, 9E9]];
	VAR robtarget OpenholeUD_6353 := [[478.45, -14.7, 180.53], [0.083709, 0.702134, 0.698657, -0.108987], [0,0,0,0], [9E9, 9E9, 9E9, 9E9, 9E9, 9E9]];
	VAR robtarget OpenholeUD_6354 := [[482.45, -14.7, 180.36], [0.096247, 0.700526, 0.696652, -0.121143], [0,0,0,0], [9E9, 9E9, 9E9, 9E9, 9E9, 9E9]];
	VAR robtarget OpenholeUD_6355 := [[486.44, -14.7, 180.2], [0.10849, 0.698734, 0.694489, -0.132985], [0,0,0,0], [9E9, 9E9, 9E9, 9E9, 9E9, 9E9]];
	VAR robtarget OpenholeUD_6356 := [[490.44, -14.7, 180.03], [0.120416, 0.696778, 0.692186, -0.144496], [0,0,0,0], [9E9, 9E9, 9E9, 9E9, 9E9, 9E9]];
	VAR robtarget OpenholeUD_6357 := [[494.44, -14.7, 179.86], [0.132007, 0.694676, 0.689761, -0.155661], [0,0,0,0], [9E9, 9E9, 9E9, 9E9, 9E9, 9E9]];
	VAR robtarget OpenholeUD_6358 := [[498.43, -14.7, 179.7], [0.14325, 0.692445, 0.687232, -0.166469], [0,0,0,0], [9E9, 9E9, 9E9, 9E9, 9E9, 9E9]];
	VAR robtarget OpenholeUD_6359 := [[502.43, -14.7, 179.53], [0.154136, 0.690103, 0.684618, -0.176914], [0,0,0,0], [9E9, 9E9, 9E9, 9E9, 9E9, 9E9]];
	VAR robtarget OpenholeUD_6360 := [[509.34, -14.7, 179.24], [0.183051, 0.683002, 0.683002, -0.183051], [0,0,0,0], [9E9, 9E9, 9E9, 9E9, 9E9, 9E9]];
	VAR robtarget OpenholeUD_6361 := [[513.34, -14.7, 179.23], [0.183051, 0.683002, 0.683002, -0.183051], [0,0,0,0], [9E9, 9E9, 9E9, 9E9, 9E9, 9E9]];
	VAR robtarget OpenholeUD_6362 := [[517.34, -14.7, 179.22], [0.183051, 0.683002, 0.683002, -0.183051], [0,0,0,0], [9E9, 9E9, 9E9, 9E9, 9E9, 9E9]];
	VAR robtarget OpenholeUD_6363 := [[521.34, -14.7, 179.21], [0.183051, 0.683002, 0.683002, -0.183051], [0,0,0,0], [9E9, 9E9, 9E9, 9E9, 9E9, 9E9]];
	VAR robtarget OpenholeUD_6364 := [[525.34, -14.7, 179.19], [0.183051, 0.683002, 0.683002, -0.183051], [0,0,0,0], [9E9, 9E9, 9E9, 9E9, 9E9, 9E9]];
	VAR robtarget OpenholeUD_6365 := [[529.34, -14.7, 179.18], [0.183051, 0.683002, 0.683002, -0.183051], [0,0,0,0], [9E9, 9E9, 9E9, 9E9, 9E9, 9E9]];
	VAR robtarget OpenholeUD_6366 := [[529.34, -14.7, 179.18], [0.183051, 0.683002, 0.683002, -0.183051], [0,0,0,0], [9E9, 9E9, 9E9, 9E9, 9E9, 9E9]];
	VAR robtarget OpenholeUD_6367 := [[529.34, -15.9, 179.87], [0.183051, 0.683002, 0.683002, -0.183051], [0,0,0,0], [9E9, 9E9, 9E9, 9E9, 9E9, 9E9]];
	VAR robtarget OpenholeUD_6368 := [[525.34, -15.9, 179.89], [0.183051, 0.683002, 0.683002, -0.183051], [0,0,0,0], [9E9, 9E9, 9E9, 9E9, 9E9, 9E9]];
	VAR robtarget OpenholeUD_6369 := [[521.34, -15.9, 179.9], [0.183051, 0.683002, 0.683002, -0.183051], [0,0,0,0], [9E9, 9E9, 9E9, 9E9, 9E9, 9E9]];
	VAR robtarget OpenholeUD_6370 := [[517.34, -15.9, 179.91], [0.183051, 0.683002, 0.683002, -0.183051], [0,0,0,0], [9E9, 9E9, 9E9, 9E9, 9E9, 9E9]];
	VAR robtarget OpenholeUD_6371 := [[513.34, -15.9, 179.92], [0.183051, 0.683002, 0.683002, -0.183051], [0,0,0,0], [9E9, 9E9, 9E9, 9E9, 9E9, 9E9]];
	VAR robtarget OpenholeUD_6372 := [[509.34, -15.9, 179.94], [0.183051, 0.683002, 0.683002, -0.183051], [0,0,0,0], [9E9, 9E9, 9E9, 9E9, 9E9, 9E9]];
	VAR robtarget OpenholeUD_6373 := [[505.34, -15.9, 180.06], [0.165348, 0.687503, 0.683592, -0.180839], [0,0,0,0], [9E9, 9E9, 9E9, 9E9, 9E9, 9E9]];
	VAR robtarget OpenholeUD_6374 := [[501.35, -15.9, 180.18], [0.154791, 0.689956, 0.686221, -0.170589], [0,0,0,0], [9E9, 9E9, 9E9, 9E9, 9E9, 9E9]];
	VAR robtarget OpenholeUD_6375 := [[497.35, -15.9, 180.3], [0.14387, 0.692316, 0.688773, -0.159975], [0,0,0,0], [9E9, 9E9, 9E9, 9E9, 9E9, 9E9]];
	VAR robtarget OpenholeUD_6376 := [[493.35, -15.9, 180.42], [0.132592, 0.694564, 0.69123, -0.149001], [0,0,0,0], [9E9, 9E9, 9E9, 9E9, 9E9, 9E9]];
	VAR robtarget OpenholeUD_6377 := [[489.35, -15.9, 180.54], [0.120965, 0.696683, 0.693575, -0.137675], [0,0,0,0], [9E9, 9E9, 9E9, 9E9, 9E9, 9E9]];
	VAR robtarget OpenholeUD_6378 := [[485.35, -15.9, 180.66], [0.109004, 0.698654, 0.695788, -0.126009], [0,0,0,0], [9E9, 9E9, 9E9, 9E9, 9E9, 9E9]];
	VAR robtarget OpenholeUD_6379 := [[481.35, -15.9, 180.78], [0.096728, 0.70046, 0.697853, -0.114021], [0,0,0,0], [9E9, 9E9, 9E9, 9E9, 9E9, 9E9]];
	VAR robtarget OpenholeUD_6380 := [[477.36, -15.9, 180.9], [0.084157, 0.702081, 0.699751, -0.101729], [0,0,0,0], [9E9, 9E9, 9E9, 9E9, 9E9, 9E9]];
	VAR robtarget OpenholeUD_6381 := [[473.36, -15.9, 181.02], [0.07132, 0.703501, 0.701463, -0.089158], [0,0,0,0], [9E9, 9E9, 9E9, 9E9, 9E9, 9E9]];
	VAR robtarget OpenholeUD_6382 := [[469.36, -15.9, 181.14], [0.058246, 0.704704, 0.702974, -0.076336], [0,0,0,0], [9E9, 9E9, 9E9, 9E9, 9E9, 9E9]];
	VAR robtarget OpenholeUD_6383 := [[465.36, -15.9, 181.26], [0.044971, 0.705675, 0.704268, -0.063297], [0,0,0,0], [9E9, 9E9, 9E9, 9E9, 9E9, 9E9]];
	VAR robtarget OpenholeUD_6384 := [[461.36, -15.9, 181.38], [0.031533, 0.706403, 0.705331, -0.050075], [0,0,0,0], [9E9, 9E9, 9E9, 9E9, 9E9, 9E9]];
	VAR robtarget OpenholeUD_6385 := [[455.21, -15.9, 181.56], [0.010638, 0.707027, 0.706492, -0.029469], [0,0,0,0], [9E9, 9E9, 9E9, 9E9, 9E9, 9E9]];
	VAR robtarget OpenholeUD_6386 := [[455.21, -15.9, 181.56], [0.010638, 0.707027, 0.706492, -0.029469], [0,0,0,0], [9E9, 9E9, 9E9, 9E9, 9E9, 9E9]];
	VAR robtarget OpenholeUD_6387 := [[455.65, -17.1, 181.62], [0.01621, 0.706921, 0.706596, -0.026879], [0,0,0,0], [9E9, 9E9, 9E9, 9E9, 9E9, 9E9]];
	VAR robtarget OpenholeUD_6388 := [[459.65, -17.1, 181.55], [0.029797, 0.706479, 0.705957, -0.040312], [0,0,0,0], [9E9, 9E9, 9E9, 9E9, 9E9, 9E9]];
	VAR robtarget OpenholeUD_6389 := [[463.65, -17.1, 181.48], [0.043274, 0.705781, 0.70507, -0.053627], [0,0,0,0], [9E9, 9E9, 9E9, 9E9, 9E9, 9E9]];
	VAR robtarget OpenholeUD_6390 := [[467.65, -17.1, 181.4], [0.056598, 0.704838, 0.703946, -0.066783], [0,0,0,0], [9E9, 9E9, 9E9, 9E9, 9E9, 9E9]];
	VAR robtarget OpenholeUD_6391 := [[471.64, -17.1, 181.33], [0.069729, 0.70366, 0.702596, -0.079741], [0,0,0,0], [9E9, 9E9, 9E9, 9E9, 9E9, 9E9]];
	VAR robtarget OpenholeUD_6392 := [[475.64, -17.1, 181.25], [0.082634, 0.702262, 0.701035, -0.092469], [0,0,0,0], [9E9, 9E9, 9E9, 9E9, 9E9, 9E9]];
	VAR robtarget OpenholeUD_6393 := [[479.64, -17.1, 181.18], [0.095277, 0.700658, 0.699277, -0.104934], [0,0,0,0], [9E9, 9E9, 9E9, 9E9, 9E9, 9E9]];
	VAR robtarget OpenholeUD_6394 := [[483.64, -17.1, 181.11], [0.107634, 0.698867, 0.697341, -0.11711], [0,0,0,0], [9E9, 9E9, 9E9, 9E9, 9E9, 9E9]];
	VAR robtarget OpenholeUD_6395 := [[487.64, -17.1, 181.03], [0.119678, 0.696905, 0.695245, -0.128976], [0,0,0,0], [9E9, 9E9, 9E9, 9E9, 9E9, 9E9]];
	VAR robtarget OpenholeUD_6396 := [[491.64, -17.1, 180.96], [0.131392, 0.694792, 0.693005, -0.140511], [0,0,0,0], [9E9, 9E9, 9E9, 9E9, 9E9, 9E9]];
	VAR robtarget OpenholeUD_6397 := [[495.64, -17.1, 180.88], [0.14276, 0.692546, 0.690642, -0.151703], [0,0,0,0], [9E9, 9E9, 9E9, 9E9, 9E9, 9E9]];
	VAR robtarget OpenholeUD_6398 := [[499.64, -17.1, 180.81], [0.153771, 0.690184, 0.688172, -0.16254], [0,0,0,0], [9E9, 9E9, 9E9, 9E9, 9E9, 9E9]];
	VAR robtarget OpenholeUD_6399 := [[503.64, -17.1, 180.73], [0.164418, 0.687726, 0.685613, -0.173015], [0,0,0,0], [9E9, 9E9, 9E9, 9E9, 9E9, 9E9]];
	VAR robtarget OpenholeUD_6400 := [[509.34, -17.1, 180.63], [0.183051, 0.683002, 0.683002, -0.183051], [0,0,0,0], [9E9, 9E9, 9E9, 9E9, 9E9, 9E9]];
	VAR robtarget OpenholeUD_6401 := [[513.34, -17.1, 180.62], [0.183051, 0.683002, 0.683002, -0.183051], [0,0,0,0], [9E9, 9E9, 9E9, 9E9, 9E9, 9E9]];
	VAR robtarget OpenholeUD_6402 := [[517.34, -17.1, 180.6], [0.183051, 0.683002, 0.683002, -0.183051], [0,0,0,0], [9E9, 9E9, 9E9, 9E9, 9E9, 9E9]];
	VAR robtarget OpenholeUD_6403 := [[521.34, -17.1, 180.59], [0.183051, 0.683002, 0.683002, -0.183051], [0,0,0,0], [9E9, 9E9, 9E9, 9E9, 9E9, 9E9]];
	VAR robtarget OpenholeUD_6404 := [[529.34, -17.1, 180.57], [0.183051, 0.683002, 0.683002, -0.183051], [0,0,0,0], [9E9, 9E9, 9E9, 9E9, 9E9, 9E9]];
	VAR robtarget OpenholeUD_6405 := [[529.34, -17.1, 180.57], [0.183051, 0.683002, 0.683002, -0.183051], [0,0,0,0], [9E9, 9E9, 9E9, 9E9, 9E9, 9E9]];
	VAR robtarget OpenholeUD_6406 := [[529.35, -18.3, 181.26], [0.183051, 0.683002, 0.683002, -0.183051], [0,0,0,0], [9E9, 9E9, 9E9, 9E9, 9E9, 9E9]];
	VAR robtarget OpenholeUD_6407 := [[525.35, -18.3, 181.27], [0.183051, 0.683002, 0.683002, -0.183051], [0,0,0,0], [9E9, 9E9, 9E9, 9E9, 9E9, 9E9]];
	VAR robtarget OpenholeUD_6408 := [[521.35, -18.3, 181.28], [0.183051, 0.683002, 0.683002, -0.183051], [0,0,0,0], [9E9, 9E9, 9E9, 9E9, 9E9, 9E9]];
	VAR robtarget OpenholeUD_6409 := [[517.35, -18.3, 181.3], [0.183051, 0.683002, 0.683002, -0.183051], [0,0,0,0], [9E9, 9E9, 9E9, 9E9, 9E9, 9E9]];
	VAR robtarget OpenholeUD_6410 := [[513.35, -18.3, 181.31], [0.183051, 0.683002, 0.683002, -0.183051], [0,0,0,0], [9E9, 9E9, 9E9, 9E9, 9E9, 9E9]];
	VAR robtarget OpenholeUD_6411 := [[509.35, -18.3, 181.32], [0.183051, 0.683002, 0.683002, -0.183051], [0,0,0,0], [9E9, 9E9, 9E9, 9E9, 9E9, 9E9]];
	VAR robtarget OpenholeUD_6412 := [[505.35, -18.3, 181.35], [0.172347, 0.685782, 0.685389, -0.173904], [0,0,0,0], [9E9, 9E9, 9E9, 9E9, 9E9, 9E9]];
	VAR robtarget OpenholeUD_6413 := [[501.35, -18.3, 181.38], [0.161924, 0.688317, 0.687941, -0.163514], [0,0,0,0], [9E9, 9E9, 9E9, 9E9, 9E9, 9E9]];
	VAR robtarget OpenholeUD_6414 := [[497.35, -18.3, 181.41], [0.151134, 0.690767, 0.690408, -0.152763], [0,0,0,0], [9E9, 9E9, 9E9, 9E9, 9E9, 9E9]];
	VAR robtarget OpenholeUD_6415 := [[493.35, -18.3, 181.43], [0.13998, 0.693113, 0.692772, -0.141657], [0,0,0,0], [9E9, 9E9, 9E9, 9E9, 9E9, 9E9]];
	VAR robtarget OpenholeUD_6416 := [[489.35, -18.3, 181.46], [0.128473, 0.695338, 0.695016, -0.130204], [0,0,0,0], [9E9, 9E9, 9E9, 9E9, 9E9, 9E9]];
	VAR robtarget OpenholeUD_6417 := [[485.35, -18.3, 181.49], [0.116625, 0.697423, 0.697121, -0.118418], [0,0,0,0], [9E9, 9E9, 9E9, 9E9, 9E9, 9E9]];
	VAR robtarget OpenholeUD_6418 := [[481.35, -18.3, 181.52], [0.104452, 0.69935, 0.699069, -0.106316], [0,0,0,0], [9E9, 9E9, 9E9, 9E9, 9E9, 9E9]];
	VAR robtarget OpenholeUD_6419 := [[477.35, -18.3, 181.55], [0.091976, 0.701099, 0.700842, -0.09392], [0,0,0,0], [9E9, 9E9, 9E9, 9E9, 9E9, 9E9]];
	VAR robtarget OpenholeUD_6420 := [[473.35, -18.3, 181.57], [0.079223, 0.702655, 0.702423, -0.081255], [0,0,0,0], [9E9, 9E9, 9E9, 9E9, 9E9, 9E9]];
	VAR robtarget OpenholeUD_6421 := [[469.35, -18.3, 181.6], [0.066221, 0.703999, 0.703795, -0.068351], [0,0,0,0], [9E9, 9E9, 9E9, 9E9, 9E9, 9E9]];
	VAR robtarget OpenholeUD_6422 := [[465.35, -18.3, 181.63], [0.053005, 0.705117, 0.704946, -0.055241], [0,0,0,0], [9E9, 9E9, 9E9, 9E9, 9E9, 9E9]];
	VAR robtarget OpenholeUD_6423 := [[461.35, -18.3, 181.66], [0.039613, 0.705996, 0.705861, -0.041962], [0,0,0,0], [9E9, 9E9, 9E9, 9E9, 9E9, 9E9]];
	VAR robtarget OpenholeUD_6424 := [[455.84, -18.3, 181.7], [0.020942, 0.706797, 0.706718, -0.023458], [0,0,0,0], [9E9, 9E9, 9E9, 9E9, 9E9, 9E9]];
	VAR robtarget OpenholeUD_6425 := [[455.84, -18.3, 181.7], [0.020942, 0.706797, 0.706718, -0.023458], [0,0,0,0], [9E9, 9E9, 9E9, 9E9, 9E9, 9E9]];
	VAR robtarget OpenholeUD_6426 := [[455.8, -19.5, 181.77], [0.024909, 0.706668, 0.706844, -0.019278], [0,0,0,0], [9E9, 9E9, 9E9, 9E9, 9E9, 9E9]];
	VAR robtarget OpenholeUD_6427 := [[459.8, -19.5, 181.79], [0.038461, 0.70606, 0.706348, -0.032741], [0,0,0,0], [9E9, 9E9, 9E9, 9E9, 9E9, 9E9]];
	VAR robtarget OpenholeUD_6428 := [[463.8, -19.5, 181.81], [0.051887, 0.7052, 0.705603, -0.046098], [0,0,0,0], [9E9, 9E9, 9E9, 9E9, 9E9, 9E9]];
	VAR robtarget OpenholeUD_6429 := [[467.8, -19.5, 181.83], [0.065145, 0.704099, 0.704615, -0.059307], [0,0,0,0], [9E9, 9E9, 9E9, 9E9, 9E9, 9E9]];
	VAR robtarget OpenholeUD_6430 := [[471.8, -19.5, 181.84], [0.078197, 0.70277, 0.703398, -0.07233], [0,0,0,0], [9E9, 9E9, 9E9, 9E9, 9E9, 9E9]];
	VAR robtarget OpenholeUD_6431 := [[475.8, -19.5, 181.86], [0.091007, 0.701226, 0.701963, -0.085133], [0,0,0,0], [9E9, 9E9, 9E9, 9E9, 9E9, 9E9]];
	VAR robtarget OpenholeUD_6432 := [[479.8, -19.5, 181.88], [0.103545, 0.699484, 0.700327, -0.097683], [0,0,0,0], [9E9, 9E9, 9E9, 9E9, 9E9, 9E9]];
	VAR robtarget OpenholeUD_6433 := [[483.8, -19.5, 181.9], [0.115784, 0.697563, 0.698506, -0.109953], [0,0,0,0], [9E9, 9E9, 9E9, 9E9, 9E9, 9E9]];
	VAR robtarget OpenholeUD_6434 := [[487.8, -19.5, 181.92], [0.127703, 0.69548, 0.696517, -0.12192], [0,0,0,0], [9E9, 9E9, 9E9, 9E9, 9E9, 9E9]];
	VAR robtarget OpenholeUD_6435 := [[491.8, -19.5, 181.93], [0.139282, 0.693254, 0.694378, -0.133563], [0,0,0,0], [9E9, 9E9, 9E9, 9E9, 9E9, 9E9]];
	VAR robtarget OpenholeUD_6436 := [[495.8, -19.5, 181.95], [0.150509, 0.690903, 0.692108, -0.144868], [0,0,0,0], [9E9, 9E9, 9E9, 9E9, 9E9, 9E9]];
	VAR robtarget OpenholeUD_6437 := [[499.8, -19.5, 181.97], [0.161375, 0.688446, 0.689724, -0.155823], [0,0,0,0], [9E9, 9E9, 9E9, 9E9, 9E9, 9E9]];
	VAR robtarget OpenholeUD_6438 := [[503.8, -19.5, 181.99], [0.171872, 0.685901, 0.687244, -0.16642], [0,0,0,0], [9E9, 9E9, 9E9, 9E9, 9E9, 9E9]];
	VAR robtarget OpenholeUD_6439 := [[509.35, -19.5, 182.01], [0.183051, 0.683002, 0.683002, -0.183051], [0,0,0,0], [9E9, 9E9, 9E9, 9E9, 9E9, 9E9]];
	VAR robtarget OpenholeUD_6440 := [[513.35, -19.5, 182], [0.183051, 0.683002, 0.683002, -0.183051], [0,0,0,0], [9E9, 9E9, 9E9, 9E9, 9E9, 9E9]];
	VAR robtarget OpenholeUD_6441 := [[517.35, -19.5, 181.99], [0.183051, 0.683002, 0.683002, -0.183051], [0,0,0,0], [9E9, 9E9, 9E9, 9E9, 9E9, 9E9]];
	VAR robtarget OpenholeUD_6442 := [[521.35, -19.5, 181.98], [0.183051, 0.683002, 0.683002, -0.183051], [0,0,0,0], [9E9, 9E9, 9E9, 9E9, 9E9, 9E9]];
	VAR robtarget OpenholeUD_6443 := [[525.35, -19.5, 181.96], [0.183051, 0.683002, 0.683002, -0.183051], [0,0,0,0], [9E9, 9E9, 9E9, 9E9, 9E9, 9E9]];
	VAR robtarget OpenholeUD_6444 := [[529.35, -19.5, 181.95], [0.183051, 0.683002, 0.683002, -0.183051], [0,0,0,0], [9E9, 9E9, 9E9, 9E9, 9E9, 9E9]];
	VAR robtarget OpenholeUD_6445 := [[529.35, -19.5, 181.95], [0.183051, 0.683002, 0.683002, -0.183051], [0,0,0,0], [9E9, 9E9, 9E9, 9E9, 9E9, 9E9]];
	VAR robtarget OpenholeUD_6446 := [[529.35, -20.7, 182.65], [0.183051, 0.683002, 0.683002, -0.183051], [0,0,0,0], [9E9, 9E9, 9E9, 9E9, 9E9, 9E9]];
	VAR robtarget OpenholeUD_6447 := [[525.35, -20.7, 182.66], [0.183051, 0.683002, 0.683002, -0.183051], [0,0,0,0], [9E9, 9E9, 9E9, 9E9, 9E9, 9E9]];
	VAR robtarget OpenholeUD_6448 := [[521.35, -20.7, 182.67], [0.183051, 0.683002, 0.683002, -0.183051], [0,0,0,0], [9E9, 9E9, 9E9, 9E9, 9E9, 9E9]];
	VAR robtarget OpenholeUD_6449 := [[517.35, -20.7, 182.68], [0.183051, 0.683002, 0.683002, -0.183051], [0,0,0,0], [9E9, 9E9, 9E9, 9E9, 9E9, 9E9]];
	VAR robtarget OpenholeUD_6450 := [[509.35, -20.7, 182.71], [0.183051, 0.683002, 0.683002, -0.183051], [0,0,0,0], [9E9, 9E9, 9E9, 9E9, 9E9, 9E9]];
	VAR robtarget OpenholeUD_6451 := [[505.35, -20.7, 182.64], [0.179333, 0.683988, 0.687114, -0.166957], [0,0,0,0], [9E9, 9E9, 9E9, 9E9, 9E9, 9E9]];
	VAR robtarget OpenholeUD_6452 := [[501.35, -20.7, 182.58], [0.169051, 0.686602, 0.689586, -0.156434], [0,0,0,0], [9E9, 9E9, 9E9, 9E9, 9E9, 9E9]];
	VAR robtarget OpenholeUD_6453 := [[497.35, -20.7, 182.51], [0.158397, 0.689137, 0.691964, -0.145553], [0,0,0,0], [9E9, 9E9, 9E9, 9E9, 9E9, 9E9]];
	VAR robtarget OpenholeUD_6454 := [[493.35, -20.7, 182.45], [0.147377, 0.691578, 0.694232, -0.134321], [0,0,0,0], [9E9, 9E9, 9E9, 9E9, 9E9, 9E9]];
	VAR robtarget OpenholeUD_6455 := [[489.35, -20.7, 182.39], [0.135997, 0.693905, 0.696371, -0.122749], [0,0,0,0], [9E9, 9E9, 9E9, 9E9, 9E9, 9E9]];
	VAR robtarget OpenholeUD_6456 := [[485.35, -20.7, 182.32], [0.124269, 0.696101, 0.698364, -0.11085], [0,0,0,0], [9E9, 9E9, 9E9, 9E9, 9E9, 9E9]];
	VAR robtarget OpenholeUD_6457 := [[481.35, -20.7, 182.26], [0.11221, 0.698147, 0.700192, -0.098644], [0,0,0,0], [9E9, 9E9, 9E9, 9E9, 9E9, 9E9]];
	VAR robtarget OpenholeUD_6458 := [[477.36, -20.7, 182.19], [0.099838, 0.700023, 0.701839, -0.086153], [0,0,0,0], [9E9, 9E9, 9E9, 9E9, 9E9, 9E9]];
	VAR robtarget OpenholeUD_6459 := [[473.36, -20.7, 182.13], [0.087177, 0.701712, 0.703287, -0.073404], [0,0,0,0], [9E9, 9E9, 9E9, 9E9, 9E9, 9E9]];
	VAR robtarget OpenholeUD_6460 := [[469.36, -20.7, 182.06], [0.074258, 0.703197, 0.70452, -0.060426], [0,0,0,0], [9E9, 9E9, 9E9, 9E9, 9E9, 9E9]];
	VAR robtarget OpenholeUD_6461 := [[465.36, -20.7, 182], [0.061112, 0.704461, 0.705526, -0.047256], [0,0,0,0], [9E9, 9E9, 9E9, 9E9, 9E9, 9E9]];
	VAR robtarget OpenholeUD_6462 := [[461.36, -20.7, 181.93], [0.047775, 0.705491, 0.706292, -0.033929], [0,0,0,0], [9E9, 9E9, 9E9, 9E9, 9E9, 9E9]];
	VAR robtarget OpenholeUD_6463 := [[455.53, -20.7, 181.84], [0.028097, 0.706548, 0.706962, -0.014326], [0,0,0,0], [9E9, 9E9, 9E9, 9E9, 9E9, 9E9]];
	VAR robtarget OpenholeUD_6464 := [[455.53, -20.7, 181.84], [0.028097, 0.706548, 0.706962, -0.014326], [0,0,0,0], [9E9, 9E9, 9E9, 9E9, 9E9, 9E9]];
	VAR robtarget OpenholeUD_6465 := [[455.01, -21.9, 181.9], [0.030395, 0.706453, 0.707056, -0.008489], [0,0,0,0], [9E9, 9E9, 9E9, 9E9, 9E9, 9E9]];
	VAR robtarget OpenholeUD_6466 := [[459, -21.9, 182.01], [0.04393, 0.705741, 0.706765, -0.021989], [0,0,0,0], [9E9, 9E9, 9E9, 9E9, 9E9, 9E9]];
	VAR robtarget OpenholeUD_6467 := [[463, -21.9, 182.12], [0.057333, 0.704779, 0.70622, -0.035406], [0,0,0,0], [9E9, 9E9, 9E9, 9E9, 9E9, 9E9]];
	VAR robtarget OpenholeUD_6468 := [[467, -21.9, 182.23], [0.070562, 0.703577, 0.705428, -0.048697], [0,0,0,0], [9E9, 9E9, 9E9, 9E9, 9E9, 9E9]];
	VAR robtarget OpenholeUD_6469 := [[471, -21.9, 182.34], [0.083579, 0.70215, 0.704399, -0.061823], [0,0,0,0], [9E9, 9E9, 9E9, 9E9, 9E9, 9E9]];
	VAR robtarget OpenholeUD_6470 := [[475, -21.9, 182.45], [0.09635, 0.700512, 0.703145, -0.074746], [0,0,0,0], [9E9, 9E9, 9E9, 9E9, 9E9, 9E9]];
	VAR robtarget OpenholeUD_6471 := [[479, -21.9, 182.56], [0.108843, 0.69868, 0.70168, -0.087435], [0,0,0,0], [9E9, 9E9, 9E9, 9E9, 9E9, 9E9]];
	VAR robtarget OpenholeUD_6472 := [[483, -21.9, 182.67], [0.121034, 0.696671, 0.70002, -0.099859], [0,0,0,0], [9E9, 9E9, 9E9, 9E9, 9E9, 9E9]];
	VAR robtarget OpenholeUD_6473 := [[486.99, -21.9, 182.78], [0.132899, 0.694506, 0.698182, -0.111992], [0,0,0,0], [9E9, 9E9, 9E9, 9E9, 9E9, 9E9]];
	VAR robtarget OpenholeUD_6474 := [[490.99, -21.9, 182.89], [0.144421, 0.692201, 0.696182, -0.123814], [0,0,0,0], [9E9, 9E9, 9E9, 9E9, 9E9, 9E9]];
	VAR robtarget OpenholeUD_6475 := [[494.99, -21.9, 183], [0.155588, 0.689777, 0.69404, -0.135307], [0,0,0,0], [9E9, 9E9, 9E9, 9E9, 9E9, 9E9]];
	VAR robtarget OpenholeUD_6476 := [[498.99, -21.9, 183.11], [0.166389, 0.687251, 0.691773, -0.146458], [0,0,0,0], [9E9, 9E9, 9E9, 9E9, 9E9, 9E9]];
	VAR robtarget OpenholeUD_6477 := [[502.99, -21.9, 183.22], [0.17682, 0.684642, 0.689399, -0.157257], [0,0,0,0], [9E9, 9E9, 9E9, 9E9, 9E9, 9E9]];
	VAR robtarget OpenholeUD_6478 := [[509.35, -21.9, 183.4], [0.183051, 0.683002, 0.683002, -0.183051], [0,0,0,0], [9E9, 9E9, 9E9, 9E9, 9E9, 9E9]];
	VAR robtarget OpenholeUD_6479 := [[513.35, -21.9, 183.39], [0.183051, 0.683002, 0.683002, -0.183051], [0,0,0,0], [9E9, 9E9, 9E9, 9E9, 9E9, 9E9]];
	VAR robtarget OpenholeUD_6480 := [[517.35, -21.9, 183.38], [0.183051, 0.683002, 0.683002, -0.183051], [0,0,0,0], [9E9, 9E9, 9E9, 9E9, 9E9, 9E9]];
	VAR robtarget OpenholeUD_6481 := [[521.35, -21.9, 183.36], [0.183051, 0.683002, 0.683002, -0.183051], [0,0,0,0], [9E9, 9E9, 9E9, 9E9, 9E9, 9E9]];
	VAR robtarget OpenholeUD_6482 := [[529.35, -21.9, 183.34], [0.183051, 0.683002, 0.683002, -0.183051], [0,0,0,0], [9E9, 9E9, 9E9, 9E9, 9E9, 9E9]];
	VAR robtarget OpenholeUD_6483 := [[529.35, -21.9, 183.34], [0.183051, 0.683002, 0.683002, -0.183051], [0,0,0,0], [9E9, 9E9, 9E9, 9E9, 9E9, 9E9]];
	VAR robtarget OpenholeUD_6484 := [[529.36, -23.1, 184.03], [0.183051, 0.683002, 0.683002, -0.183051], [0,0,0,0], [9E9, 9E9, 9E9, 9E9, 9E9, 9E9]];
	VAR robtarget OpenholeUD_6485 := [[525.36, -23.1, 184.04], [0.183051, 0.683002, 0.683002, -0.183051], [0,0,0,0], [9E9, 9E9, 9E9, 9E9, 9E9, 9E9]];
	VAR robtarget OpenholeUD_6486 := [[521.36, -23.1, 184.06], [0.183051, 0.683002, 0.683002, -0.183051], [0,0,0,0], [9E9, 9E9, 9E9, 9E9, 9E9, 9E9]];
	VAR robtarget OpenholeUD_6487 := [[517.36, -23.1, 184.07], [0.183051, 0.683002, 0.683002, -0.183051], [0,0,0,0], [9E9, 9E9, 9E9, 9E9, 9E9, 9E9]];
	VAR robtarget OpenholeUD_6488 := [[513.36, -23.1, 184.08], [0.183051, 0.683002, 0.683002, -0.183051], [0,0,0,0], [9E9, 9E9, 9E9, 9E9, 9E9, 9E9]];
	VAR robtarget OpenholeUD_6489 := [[509.36, -23.1, 184.09], [0.183051, 0.683002, 0.683002, -0.183051], [0,0,0,0], [9E9, 9E9, 9E9, 9E9, 9E9, 9E9]];
	VAR robtarget OpenholeUD_6490 := [[505.36, -23.1, 183.94], [0.1863, 0.682123, 0.688766, -0.160004], [0,0,0,0], [9E9, 9E9, 9E9, 9E9, 9E9, 9E9]];
	VAR robtarget OpenholeUD_6491 := [[501.36, -23.1, 183.78], [0.176163, 0.684811, 0.691154, -0.149355], [0,0,0,0], [9E9, 9E9, 9E9, 9E9, 9E9, 9E9]];
	VAR robtarget OpenholeUD_6492 := [[497.36, -23.1, 183.62], [0.165653, 0.687429, 0.69344, -0.138351], [0,0,0,0], [9E9, 9E9, 9E9, 9E9, 9E9, 9E9]];
	VAR robtarget OpenholeUD_6493 := [[493.37, -23.1, 183.47], [0.154773, 0.68996, 0.695608, -0.127002], [0,0,0,0], [9E9, 9E9, 9E9, 9E9, 9E9, 9E9]];
	VAR robtarget OpenholeUD_6494 := [[489.37, -23.1, 183.31], [0.143528, 0.692387, 0.69764, -0.115318], [0,0,0,0], [9E9, 9E9, 9E9, 9E9, 9E9, 9E9]];
	VAR robtarget OpenholeUD_6495 := [[485.37, -23.1, 183.15], [0.131929, 0.69469, 0.699518, -0.103316], [0,0,0,0], [9E9, 9E9, 9E9, 9E9, 9E9, 9E9]];
	VAR robtarget OpenholeUD_6496 := [[481.38, -23.1, 183], [0.119991, 0.696852, 0.701225, -0.091014], [0,0,0,0], [9E9, 9E9, 9E9, 9E9, 9E9, 9E9]];
	VAR robtarget OpenholeUD_6497 := [[477.38, -23.1, 182.84], [0.107731, 0.698852, 0.702743, -0.078437], [0,0,0,0], [9E9, 9E9, 9E9, 9E9, 9E9, 9E9]];
	VAR robtarget OpenholeUD_6498 := [[473.38, -23.1, 182.68], [0.095174, 0.700672, 0.704056, -0.065612], [0,0,0,0], [9E9, 9E9, 9E9, 9E9, 9E9, 9E9]];
	VAR robtarget OpenholeUD_6499 := [[469.39, -23.1, 182.53], [0.082346, 0.702296, 0.70515, -0.052571], [0,0,0,0], [9E9, 9E9, 9E9, 9E9, 9E9, 9E9]];
	VAR robtarget OpenholeUD_6500 := [[465.39, -23.1, 182.37], [0.069279, 0.703705, 0.706011, -0.039349], [0,0,0,0], [9E9, 9E9, 9E9, 9E9, 9E9, 9E9]];
	VAR robtarget OpenholeUD_6501 := [[461.39, -23.1, 182.21], [0.056008, 0.704885, 0.706629, -0.025984], [0,0,0,0], [9E9, 9E9, 9E9, 9E9, 9E9, 9E9]];
	VAR robtarget OpenholeUD_6502 := [[454.13, -23.1, 181.93], [0.031514, 0.706404, 0.707105, -0.001479], [0,0,0,0], [9E9, 9E9, 9E9, 9E9, 9E9, 9E9]];
	VAR robtarget OpenholeUD_6503 := [[454.13, -23.1, 181.93], [0.031514, 0.706404, 0.707105, -0.001479], [0,0,0,0], [9E9, 9E9, 9E9, 9E9, 9E9, 9E9]];
	VAR robtarget OpenholeUD_6504 := [[452.65, -24.3, 181.91], [0.030549, 0.706447, 0.707066, 0.007602], [0,0,0,0], [9E9, 9E9, 9E9, 9E9, 9E9, 9E9]];
	VAR robtarget OpenholeUD_6505 := [[456.64, -24.3, 182.11], [0.044105, 0.70573, 0.707082, -0.00593], [0,0,0,0], [9E9, 9E9, 9E9, 9E9, 9E9, 9E9]];
	VAR robtarget OpenholeUD_6506 := [[460.64, -24.3, 182.31], [0.057539, 0.704762, 0.70684, -0.01942], [0,0,0,0], [9E9, 9E9, 9E9, 9E9, 9E9, 9E9]];
	VAR robtarget OpenholeUD_6507 := [[464.63, -24.3, 182.52], [0.07081, 0.703552, 0.706345, -0.032822], [0,0,0,0], [9E9, 9E9, 9E9, 9E9, 9E9, 9E9]];
	VAR robtarget OpenholeUD_6508 := [[468.63, -24.3, 182.72], [0.083878, 0.702114, 0.705603, -0.046096], [0,0,0,0], [9E9, 9E9, 9E9, 9E9, 9E9, 9E9]];
	VAR robtarget OpenholeUD_6509 := [[472.62, -24.3, 182.92], [0.096707, 0.700463, 0.704624, -0.059203], [0,0,0,0], [9E9, 9E9, 9E9, 9E9, 9E9, 9E9]];
	VAR robtarget OpenholeUD_6510 := [[476.62, -24.3, 183.13], [0.109266, 0.698614, 0.703421, -0.072106], [0,0,0,0], [9E9, 9E9, 9E9, 9E9, 9E9, 9E9]];
	VAR robtarget OpenholeUD_6511 := [[480.61, -24.3, 183.33], [0.121527, 0.696585, 0.702007, -0.084772], [0,0,0,0], [9E9, 9E9, 9E9, 9E9, 9E9, 9E9]];
	VAR robtarget OpenholeUD_6512 := [[484.61, -24.3, 183.53], [0.133467, 0.694397, 0.700398, -0.097173], [0,0,0,0], [9E9, 9E9, 9E9, 9E9, 9E9, 9E9]];
	VAR robtarget OpenholeUD_6513 := [[488.6, -24.3, 183.73], [0.145066, 0.692066, 0.698611, -0.109283], [0,0,0,0], [9E9, 9E9, 9E9, 9E9, 9E9, 9E9]];
	VAR robtarget OpenholeUD_6514 := [[492.6, -24.3, 183.94], [0.156312, 0.689613, 0.696663, -0.121082], [0,0,0,0], [9E9, 9E9, 9E9, 9E9, 9E9, 9E9]];
	VAR robtarget OpenholeUD_6515 := [[496.59, -24.3, 184.14], [0.167192, 0.687057, 0.694572, -0.132553], [0,0,0,0], [9E9, 9E9, 9E9, 9E9, 9E9, 9E9]];
	VAR robtarget OpenholeUD_6516 := [[500.59, -24.3, 184.34], [0.177701, 0.684414, 0.692355, -0.143683], [0,0,0,0], [9E9, 9E9, 9E9, 9E9, 9E9, 9E9]];
	VAR robtarget OpenholeUD_6517 := [[504.58, -24.3, 184.54], [0.187836, 0.681702, 0.69003, -0.154462], [0,0,0,0], [9E9, 9E9, 9E9, 9E9, 9E9, 9E9]];
	VAR robtarget OpenholeUD_6518 := [[509.36, -24.3, 184.79], [0.183051, 0.683002, 0.683002, -0.183051], [0,0,0,0], [9E9, 9E9, 9E9, 9E9, 9E9, 9E9]];
	VAR robtarget OpenholeUD_6519 := [[513.36, -24.3, 184.77], [0.183051, 0.683002, 0.683002, -0.183051], [0,0,0,0], [9E9, 9E9, 9E9, 9E9, 9E9, 9E9]];
	VAR robtarget OpenholeUD_6520 := [[517.36, -24.3, 184.76], [0.183051, 0.683002, 0.683002, -0.183051], [0,0,0,0], [9E9, 9E9, 9E9, 9E9, 9E9, 9E9]];
	VAR robtarget OpenholeUD_6521 := [[521.36, -24.3, 184.75], [0.183051, 0.683002, 0.683002, -0.183051], [0,0,0,0], [9E9, 9E9, 9E9, 9E9, 9E9, 9E9]];
	VAR robtarget OpenholeUD_6522 := [[525.36, -24.3, 184.74], [0.183051, 0.683002, 0.683002, -0.183051], [0,0,0,0], [9E9, 9E9, 9E9, 9E9, 9E9, 9E9]];
	VAR robtarget OpenholeUD_6523 := [[529.36, -24.3, 184.72], [0.183051, 0.683002, 0.683002, -0.183051], [0,0,0,0], [9E9, 9E9, 9E9, 9E9, 9E9, 9E9]];
	VAR robtarget OpenholeUD_6524 := [[529.35, -20.84, 182.72], [0.183051, 0.683002, 0.683002, -0.183051], [0,0,0,0], [9E9, 9E9, 9E9, 9E9, 9E9, 9E9]];
	VAR robtarget OpenholeUD_6525 := [[529.34, -17.37, 180.72], [0.183051, 0.683002, 0.683002, -0.183051], [0,0,0,0], [9E9, 9E9, 9E9, 9E9, 9E9, 9E9]];
	VAR robtarget OpenholeUD_6526 := [[529.33, -11.1, 177.1], [0.183051, 0.683002, 0.683002, -0.183051], [0,0,0,0], [9E9, 9E9, 9E9, 9E9, 9E9, 9E9]];
	VAR robtarget OpenholeUD_6527 := [[525.33, -11.1, 177.11], [0.183051, 0.683002, 0.683002, -0.183051], [0,0,0,0], [9E9, 9E9, 9E9, 9E9, 9E9, 9E9]];
	VAR robtarget OpenholeUD_6528 := [[521.33, -11.1, 177.13], [0.183051, 0.683002, 0.683002, -0.183051], [0,0,0,0], [9E9, 9E9, 9E9, 9E9, 9E9, 9E9]];
	VAR robtarget OpenholeUD_6529 := [[517.33, -11.1, 177.14], [0.183051, 0.683002, 0.683002, -0.183051], [0,0,0,0], [9E9, 9E9, 9E9, 9E9, 9E9, 9E9]];
	VAR robtarget OpenholeUD_6530 := [[513.33, -11.1, 177.15], [0.183051, 0.683002, 0.683002, -0.183051], [0,0,0,0], [9E9, 9E9, 9E9, 9E9, 9E9, 9E9]];
	VAR robtarget OpenholeUD_6531 := [[509.33, -11.1, 177.16], [0.183051, 0.683002, 0.683002, -0.183051], [0,0,0,0], [9E9, 9E9, 9E9, 9E9, 9E9, 9E9]];
	VAR robtarget OpenholeUD_6532 := [[505.35, -11.1, 177.47], [0.151337, 0.690722, 0.679789, -0.194646], [0,0,0,0], [9E9, 9E9, 9E9, 9E9, 9E9, 9E9]];
	VAR robtarget OpenholeUD_6533 := [[501.36, -11.1, 177.77], [0.140534, 0.693001, 0.68256, -0.184693], [0,0,0,0], [9E9, 9E9, 9E9, 9E9, 9E9, 9E9]];
	VAR robtarget OpenholeUD_6534 := [[497.37, -11.1, 178.08], [0.129376, 0.69517, 0.68527, -0.17437], [0,0,0,0], [9E9, 9E9, 9E9, 9E9, 9E9, 9E9]];
	VAR robtarget OpenholeUD_6535 := [[493.38, -11.1, 178.38], [0.117871, 0.697213, 0.687902, -0.16368], [0,0,0,0], [9E9, 9E9, 9E9, 9E9, 9E9, 9E9]];
	VAR robtarget OpenholeUD_6536 := [[489.39, -11.1, 178.69], [0.106032, 0.699112, 0.690438, -0.15263], [0,0,0,0], [9E9, 9E9, 9E9, 9E9, 9E9, 9E9]];
	VAR robtarget OpenholeUD_6537 := [[485.4, -11.1, 178.99], [0.093873, 0.700848, 0.69286, -0.141228], [0,0,0,0], [9E9, 9E9, 9E9, 9E9, 9E9, 9E9]];
	VAR robtarget OpenholeUD_6538 := [[481.41, -11.1, 179.29], [0.081417, 0.702404, 0.695149, -0.129489], [0,0,0,0], [9E9, 9E9, 9E9, 9E9, 9E9, 9E9]];
	VAR robtarget OpenholeUD_6539 := [[477.43, -11.1, 179.6], [0.068686, 0.703763, 0.697288, -0.11743], [0,0,0,0], [9E9, 9E9, 9E9, 9E9, 9E9, 9E9]];
	VAR robtarget OpenholeUD_6540 := [[473.44, -11.1, 179.9], [0.05571, 0.704909, 0.699256, -0.105073], [0,0,0,0], [9E9, 9E9, 9E9, 9E9, 9E9, 9E9]];
	VAR robtarget OpenholeUD_6541 := [[469.45, -11.1, 180.21], [0.042522, 0.705827, 0.701038, -0.092444], [0,0,0,0], [9E9, 9E9, 9E9, 9E9, 9E9, 9E9]];
	VAR robtarget OpenholeUD_6542 := [[465.46, -11.1, 180.51], [0.029158, 0.706505, 0.702615, -0.079573], [0,0,0,0], [9E9, 9E9, 9E9, 9E9, 9E9, 9E9]];
	VAR robtarget OpenholeUD_6543 := [[461.47, -11.1, 180.82], [0.015658, 0.706933, 0.703973, -0.066494], [0,0,0,0], [9E9, 9E9, 9E9, 9E9, 9E9, 9E9]];
	VAR robtarget OpenholeUD_6544 := [[457.48, -11.1, 181.12], [0.002064, 0.707104, 0.705099, -0.053243], [0,0,0,0], [9E9, 9E9, 9E9, 9E9, 9E9, 9E9]];
	VAR robtarget OpenholeUD_6545 := [[453.5, -11.1, 181.42], [-0.011579, 0.707012, 0.705982, -0.039862], [0,0,0,0], [9E9, 9E9, 9E9, 9E9, 9E9, 9E9]];
	VAR robtarget OpenholeUD_6546 := [[449.51, -11.1, 181.73], [-0.025225, 0.706657, 0.706614, -0.026391], [0,0,0,0], [9E9, 9E9, 9E9, 9E9, 9E9, 9E9]];
	VAR robtarget OpenholeUD_6547 := [[445.52, -11.1, 182.03], [-0.038829, 0.70604, 0.70699, -0.012875], [0,0,0,0], [9E9, 9E9, 9E9, 9E9, 9E9, 9E9]];
	VAR robtarget OpenholeUD_6548 := [[441.53, -11.1, 182.34], [-0.052344, 0.705167, 0.707106, 0.000643], [0,0,0,0], [9E9, 9E9, 9E9, 9E9, 9E9, 9E9]];
	VAR robtarget OpenholeUD_6549 := [[437.54, -11.1, 182.64], [-0.065728, 0.704045, 0.706966, 0.014118], [0,0,0,0], [9E9, 9E9, 9E9, 9E9, 9E9, 9E9]];
	VAR robtarget OpenholeUD_6550 := [[433.55, -11.1, 182.95], [-0.078938, 0.702687, 0.706572, 0.027508], [0,0,0,0], [9E9, 9E9, 9E9, 9E9, 9E9, 9E9]];
	VAR robtarget OpenholeUD_6551 := [[429.57, -11.1, 183.25], [-0.091936, 0.701105, 0.70593, 0.040772], [0,0,0,0], [9E9, 9E9, 9E9, 9E9, 9E9, 9E9]];
	VAR robtarget OpenholeUD_6552 := [[425.58, -11.1, 183.56], [-0.104687, 0.699314, 0.705052, 0.053869], [0,0,0,0], [9E9, 9E9, 9E9, 9E9, 9E9, 9E9]];
	VAR robtarget OpenholeUD_6553 := [[421.59, -11.1, 183.86], [-0.117158, 0.697333, 0.703948, 0.066766], [0,0,0,0], [9E9, 9E9, 9E9, 9E9, 9E9, 9E9]];
	VAR robtarget OpenholeUD_6554 := [[417.6, -11.1, 184.16], [-0.129325, 0.69518, 0.702631, 0.079429], [0,0,0,0], [9E9, 9E9, 9E9, 9E9, 9E9, 9E9]];
	VAR robtarget OpenholeUD_6555 := [[413.61, -11.1, 184.47], [-0.141163, 0.692873, 0.701118, 0.091831], [0,0,0,0], [9E9, 9E9, 9E9, 9E9, 9E9, 9E9]];
	VAR robtarget OpenholeUD_6556 := [[409.62, -11.1, 184.77], [-0.152655, 0.690432, 0.699425, 0.103945], [0,0,0,0], [9E9, 9E9, 9E9, 9E9, 9E9, 9E9]];
	VAR robtarget OpenholeUD_6557 := [[405.63, -11.1, 185.08], [-0.163787, 0.687876, 0.697568, 0.115753], [0,0,0,0], [9E9, 9E9, 9E9, 9E9, 9E9, 9E9]];
	VAR robtarget OpenholeUD_6558 := [[401.65, -11.1, 185.38], [-0.17455, 0.685224, 0.695565, 0.127237], [0,0,0,0], [9E9, 9E9, 9E9, 9E9, 9E9, 9E9]];
	VAR robtarget OpenholeUD_6559 := [[397.66, -11.1, 185.69], [-0.184937, 0.682494, 0.693433, 0.138384], [0,0,0,0], [9E9, 9E9, 9E9, 9E9, 9E9, 9E9]];
	VAR robtarget OpenholeUD_6560 := [[393.67, -11.1, 185.99], [-0.194947, 0.679703, 0.69119, 0.149185], [0,0,0,0], [9E9, 9E9, 9E9, 9E9, 9E9, 9E9]];
	VAR robtarget OpenholeUD_6561 := [[389.36, -11.1, 186.32], [-0.205335, 0.676637, 0.688661, 0.160457], [0,0,0,0], [9E9, 9E9, 9E9, 9E9, 9E9, 9E9]];
	VAR robtarget OpenholeUD_6562 := [[385.36, -11.1, 186.33], [-0.183051, 0.683002, 0.683002, 0.183051], [0,0,0,0], [9E9, 9E9, 9E9, 9E9, 9E9, 9E9]];
	VAR robtarget OpenholeUD_6563 := [[381.36, -11.1, 186.34], [-0.183051, 0.683002, 0.683002, 0.183051], [0,0,0,0], [9E9, 9E9, 9E9, 9E9, 9E9, 9E9]];
	VAR robtarget OpenholeUD_6564 := [[377.36, -11.1, 186.36], [-0.183051, 0.683002, 0.683002, 0.183051], [0,0,0,0], [9E9, 9E9, 9E9, 9E9, 9E9, 9E9]];
	VAR robtarget OpenholeUD_6565 := [[373.36, -11.1, 186.37], [-0.183051, 0.683002, 0.683002, 0.183051], [0,0,0,0], [9E9, 9E9, 9E9, 9E9, 9E9, 9E9]];
	VAR robtarget OpenholeUD_6566 := [[369.36, -11.1, 186.38], [-0.183051, 0.683002, 0.683002, 0.183051], [0,0,0,0], [9E9, 9E9, 9E9, 9E9, 9E9, 9E9]];
	VAR robtarget OpenholeUD_6567 := [[369.36, -11.1, 186.38], [-0.183051, 0.683002, 0.683002, 0.183051], [0,0,0,0], [9E9, 9E9, 9E9, 9E9, 9E9, 9E9]];
	VAR robtarget OpenholeUD_6568 := [[369.36, -9.9, 187.07], [-0.183051, 0.683002, 0.683002, 0.183051], [0,0,0,0], [9E9, 9E9, 9E9, 9E9, 9E9, 9E9]];
	VAR robtarget OpenholeUD_6569 := [[373.36, -9.9, 187.06], [-0.183051, 0.683002, 0.683002, 0.183051], [0,0,0,0], [9E9, 9E9, 9E9, 9E9, 9E9, 9E9]];
	VAR robtarget OpenholeUD_6570 := [[377.36, -9.9, 187.05], [-0.183051, 0.683002, 0.683002, 0.183051], [0,0,0,0], [9E9, 9E9, 9E9, 9E9, 9E9, 9E9]];
	VAR robtarget OpenholeUD_6571 := [[381.36, -9.9, 187.04], [-0.183051, 0.683002, 0.683002, 0.183051], [0,0,0,0], [9E9, 9E9, 9E9, 9E9, 9E9, 9E9]];
	VAR robtarget OpenholeUD_6572 := [[385.36, -9.9, 187.02], [-0.183051, 0.683002, 0.683002, 0.183051], [0,0,0,0], [9E9, 9E9, 9E9, 9E9, 9E9, 9E9]];
	VAR robtarget OpenholeUD_6573 := [[389.36, -9.9, 187.01], [-0.208708, 0.675604, 0.689448, 0.157038], [0,0,0,0], [9E9, 9E9, 9E9, 9E9, 9E9, 9E9]];
	VAR robtarget OpenholeUD_6574 := [[393.35, -9.9, 186.66], [-0.199185, 0.678473, 0.691752, 0.146559], [0,0,0,0], [9E9, 9E9, 9E9, 9E9, 9E9, 9E9]];
	VAR robtarget OpenholeUD_6575 := [[397.33, -9.9, 186.31], [-0.189285, 0.681301, 0.693958, 0.135731], [0,0,0,0], [9E9, 9E9, 9E9, 9E9, 9E9, 9E9]];
	VAR robtarget OpenholeUD_6576 := [[401.32, -9.9, 185.96], [-0.179005, 0.684074, 0.69605, 0.124559], [0,0,0,0], [9E9, 9E9, 9E9, 9E9, 9E9, 9E9]];
	VAR robtarget OpenholeUD_6577 := [[405.3, -9.9, 185.61], [-0.168349, 0.686774, 0.698011, 0.113052], [0,0,0,0], [9E9, 9E9, 9E9, 9E9, 9E9, 9E9]];
	VAR robtarget OpenholeUD_6578 := [[409.29, -9.9, 185.26], [-0.157321, 0.689384, 0.699824, 0.101224], [0,0,0,0], [9E9, 9E9, 9E9, 9E9, 9E9, 9E9]];
	VAR robtarget OpenholeUD_6579 := [[413.27, -9.9, 184.91], [-0.145929, 0.691885, 0.701472, 0.089091], [0,0,0,0], [9E9, 9E9, 9E9, 9E9, 9E9, 9E9]];
	VAR robtarget OpenholeUD_6580 := [[417.26, -9.9, 184.56], [-0.134187, 0.694258, 0.702937, 0.076674], [0,0,0,0], [9E9, 9E9, 9E9, 9E9, 9E9, 9E9]];
	VAR robtarget OpenholeUD_6581 := [[421.24, -9.9, 184.21], [-0.122111, 0.696483, 0.704205, 0.063998], [0,0,0,0], [9E9, 9E9, 9E9, 9E9, 9E9, 9E9]];
	VAR robtarget OpenholeUD_6582 := [[425.23, -9.9, 183.86], [-0.109724, 0.698542, 0.705259, 0.051092], [0,0,0,0], [9E9, 9E9, 9E9, 9E9, 9E9, 9E9]];
	VAR robtarget OpenholeUD_6583 := [[429.21, -9.9, 183.51], [-0.09705, 0.700415, 0.706086, 0.037987], [0,0,0,0], [9E9, 9E9, 9E9, 9E9, 9E9, 9E9]];
	VAR robtarget OpenholeUD_6584 := [[433.19, -9.9, 183.16], [-0.08412, 0.702085, 0.706675, 0.024721], [0,0,0,0], [9E9, 9E9, 9E9, 9E9, 9E9, 9E9]];
	VAR robtarget OpenholeUD_6585 := [[437.18, -9.9, 182.81], [-0.070968, 0.703536, 0.707016, 0.01133], [0,0,0,0], [9E9, 9E9, 9E9, 9E9, 9E9, 9E9]];
	VAR robtarget OpenholeUD_6586 := [[441.16, -9.9, 182.46], [-0.057633, 0.704754, 0.707104, -0.002142], [0,0,0,0], [9E9, 9E9, 9E9, 9E9, 9E9, 9E9]];
	VAR robtarget OpenholeUD_6587 := [[445.15, -9.9, 182.11], [-0.044154, 0.705727, 0.706933, -0.015654], [0,0,0,0], [9E9, 9E9, 9E9, 9E9, 9E9, 9E9]];
	VAR robtarget OpenholeUD_6588 := [[449.13, -9.9, 181.76], [-0.030577, 0.706445, 0.706505, -0.029161], [0,0,0,0], [9E9, 9E9, 9E9, 9E9, 9E9, 9E9]];
	VAR robtarget OpenholeUD_6589 := [[453.12, -9.9, 181.41], [-0.016945, 0.706904, 0.705821, -0.04262], [0,0,0,0], [9E9, 9E9, 9E9, 9E9, 9E9, 9E9]];
	VAR robtarget OpenholeUD_6590 := [[457.1, -9.9, 181.06], [-0.003305, 0.707099, 0.704887, -0.055986], [0,0,0,0], [9E9, 9E9, 9E9, 9E9, 9E9, 9E9]];
	VAR robtarget OpenholeUD_6591 := [[461.09, -9.9, 180.71], [0.010298, 0.707032, 0.703711, -0.069219], [0,0,0,0], [9E9, 9E9, 9E9, 9E9, 9E9, 9E9]];
	VAR robtarget OpenholeUD_6592 := [[465.07, -9.9, 180.36], [0.023819, 0.706705, 0.702304, -0.082278], [0,0,0,0], [9E9, 9E9, 9E9, 9E9, 9E9, 9E9]];
	VAR robtarget OpenholeUD_6593 := [[469.06, -9.9, 180.01], [0.037215, 0.706127, 0.700679, -0.095126], [0,0,0,0], [9E9, 9E9, 9E9, 9E9, 9E9, 9E9]];
	VAR robtarget OpenholeUD_6594 := [[473.04, -9.9, 179.66], [0.050446, 0.705305, 0.698852, -0.107729], [0,0,0,0], [9E9, 9E9, 9E9, 9E9, 9E9, 9E9]];
	VAR robtarget OpenholeUD_6595 := [[477.03, -9.9, 179.31], [0.063474, 0.704252, 0.69684, -0.120059], [0,0,0,0], [9E9, 9E9, 9E9, 9E9, 9E9, 9E9]];
	VAR robtarget OpenholeUD_6596 := [[481.01, -9.9, 178.96], [0.076265, 0.702982, 0.69466, -0.132088], [0,0,0,0], [9E9, 9E9, 9E9, 9E9, 9E9, 9E9]];
	VAR robtarget OpenholeUD_6597 := [[485, -9.9, 178.61], [0.088791, 0.70151, 0.692331, -0.143796], [0,0,0,0], [9E9, 9E9, 9E9, 9E9, 9E9, 9E9]];
	VAR robtarget OpenholeUD_6598 := [[488.98, -9.9, 178.26], [0.101026, 0.699853, 0.689872, -0.155164], [0,0,0,0], [9E9, 9E9, 9E9, 9E9, 9E9, 9E9]];
	VAR robtarget OpenholeUD_6599 := [[492.96, -9.9, 177.91], [0.112948, 0.698028, 0.687302, -0.16618], [0,0,0,0], [9E9, 9E9, 9E9, 9E9, 9E9, 9E9]];
	VAR robtarget OpenholeUD_6600 := [[496.95, -9.9, 177.56], [0.12454, 0.696053, 0.684638, -0.176835], [0,0,0,0], [9E9, 9E9, 9E9, 9E9, 9E9, 9E9]];
	VAR robtarget OpenholeUD_6601 := [[500.93, -9.9, 177.21], [0.13579, 0.693946, 0.681899, -0.187121], [0,0,0,0], [9E9, 9E9, 9E9, 9E9, 9E9, 9E9]];
	VAR robtarget OpenholeUD_6602 := [[504.92, -9.9, 176.86], [0.146688, 0.691724, 0.6791, -0.197037], [0,0,0,0], [9E9, 9E9, 9E9, 9E9, 9E9, 9E9]];
	VAR robtarget OpenholeUD_6603 := [[509.33, -9.9, 176.47], [0.183051, 0.683002, 0.683002, -0.183051], [0,0,0,0], [9E9, 9E9, 9E9, 9E9, 9E9, 9E9]];
	VAR robtarget OpenholeUD_6604 := [[513.33, -9.9, 176.46], [0.183051, 0.683002, 0.683002, -0.183051], [0,0,0,0], [9E9, 9E9, 9E9, 9E9, 9E9, 9E9]];
	VAR robtarget OpenholeUD_6605 := [[517.33, -9.9, 176.45], [0.183051, 0.683002, 0.683002, -0.183051], [0,0,0,0], [9E9, 9E9, 9E9, 9E9, 9E9, 9E9]];
	VAR robtarget OpenholeUD_6606 := [[521.33, -9.9, 176.43], [0.183051, 0.683002, 0.683002, -0.183051], [0,0,0,0], [9E9, 9E9, 9E9, 9E9, 9E9, 9E9]];
	VAR robtarget OpenholeUD_6607 := [[529.33, -9.9, 176.41], [0.183051, 0.683002, 0.683002, -0.183051], [0,0,0,0], [9E9, 9E9, 9E9, 9E9, 9E9, 9E9]];
	VAR robtarget OpenholeUD_6608 := [[529.33, -9.9, 176.41], [0.183051, 0.683002, 0.683002, -0.183051], [0,0,0,0], [9E9, 9E9, 9E9, 9E9, 9E9, 9E9]];
	VAR robtarget OpenholeUD_6609 := [[529.33, -8.7, 175.72], [0.183051, 0.683002, 0.683002, -0.183051], [0,0,0,0], [9E9, 9E9, 9E9, 9E9, 9E9, 9E9]];
	VAR robtarget OpenholeUD_6610 := [[525.33, -8.7, 175.73], [0.183051, 0.683002, 0.683002, -0.183051], [0,0,0,0], [9E9, 9E9, 9E9, 9E9, 9E9, 9E9]];
	VAR robtarget OpenholeUD_6611 := [[521.33, -8.7, 175.74], [0.183051, 0.683002, 0.683002, -0.183051], [0,0,0,0], [9E9, 9E9, 9E9, 9E9, 9E9, 9E9]];
	VAR robtarget OpenholeUD_6612 := [[517.33, -8.7, 175.75], [0.183051, 0.683002, 0.683002, -0.183051], [0,0,0,0], [9E9, 9E9, 9E9, 9E9, 9E9, 9E9]];
	VAR robtarget OpenholeUD_6613 := [[509.33, -8.7, 175.78], [0.183051, 0.683002, 0.683002, -0.183051], [0,0,0,0], [9E9, 9E9, 9E9, 9E9, 9E9, 9E9]];
	VAR robtarget OpenholeUD_6614 := [[505.35, -8.7, 176.17], [0.14434, 0.692218, 0.677787, -0.201505], [0,0,0,0], [9E9, 9E9, 9E9, 9E9, 9E9, 9E9]];
	VAR robtarget OpenholeUD_6615 := [[501.37, -8.7, 176.57], [0.133425, 0.694405, 0.680623, -0.191707], [0,0,0,0], [9E9, 9E9, 9E9, 9E9, 9E9, 9E9]];
	VAR robtarget OpenholeUD_6616 := [[497.39, -8.7, 176.97], [0.122161, 0.696474, 0.683406, -0.181538], [0,0,0,0], [9E9, 9E9, 9E9, 9E9, 9E9, 9E9]];
	VAR robtarget OpenholeUD_6617 := [[493.41, -8.7, 177.36], [0.110556, 0.698411, 0.686119, -0.170999], [0,0,0,0], [9E9, 9E9, 9E9, 9E9, 9E9, 9E9]];
	VAR robtarget OpenholeUD_6618 := [[489.43, -8.7, 177.76], [0.098623, 0.700195, 0.688745, -0.160096], [0,0,0,0], [9E9, 9E9, 9E9, 9E9, 9E9, 9E9]];
	VAR robtarget OpenholeUD_6619 := [[485.45, -8.7, 178.15], [0.08638, 0.701811, 0.691265, -0.148837], [0,0,0,0], [9E9, 9E9, 9E9, 9E9, 9E9, 9E9]];
	VAR robtarget OpenholeUD_6620 := [[481.47, -8.7, 178.55], [0.073848, 0.70324, 0.693662, -0.137233], [0,0,0,0], [9E9, 9E9, 9E9, 9E9, 9E9, 9E9]];
	VAR robtarget OpenholeUD_6621 := [[477.49, -8.7, 178.94], [0.061052, 0.704466, 0.695916, -0.125303], [0,0,0,0], [9E9, 9E9, 9E9, 9E9, 9E9, 9E9]];
	VAR robtarget OpenholeUD_6622 := [[473.51, -8.7, 179.34], [0.048022, 0.705474, 0.698009, -0.113065], [0,0,0,0], [9E9, 9E9, 9E9, 9E9, 9E9, 9E9]];
	VAR robtarget OpenholeUD_6623 := [[469.53, -8.7, 179.74], [0.034792, 0.70625, 0.699922, -0.100545], [0,0,0,0], [9E9, 9E9, 9E9, 9E9, 9E9, 9E9]];
	VAR robtarget OpenholeUD_6624 := [[465.54, -8.7, 180.13], [0.021398, 0.706783, 0.701638, -0.087772], [0,0,0,0], [9E9, 9E9, 9E9, 9E9, 9E9, 9E9]];
	VAR robtarget OpenholeUD_6625 := [[461.56, -8.7, 180.53], [0.007882, 0.707063, 0.703142, -0.074778], [0,0,0,0], [9E9, 9E9, 9E9, 9E9, 9E9, 9E9]];
	VAR robtarget OpenholeUD_6626 := [[457.58, -8.7, 180.92], [-0.005715, 0.707084, 0.704419, -0.061599], [0,0,0,0], [9E9, 9E9, 9E9, 9E9, 9E9, 9E9]];
	VAR robtarget OpenholeUD_6627 := [[453.6, -8.7, 181.32], [-0.019347, 0.706842, 0.705457, -0.048275], [0,0,0,0], [9E9, 9E9, 9E9, 9E9, 9E9, 9E9]];
	VAR robtarget OpenholeUD_6628 := [[449.62, -8.7, 181.71], [-0.032968, 0.706338, 0.706248, -0.034846], [0,0,0,0], [9E9, 9E9, 9E9, 9E9, 9E9, 9E9]];
	VAR robtarget OpenholeUD_6629 := [[445.64, -8.7, 182.11], [-0.046534, 0.705574, 0.706784, -0.021357], [0,0,0,0], [9E9, 9E9, 9E9, 9E9, 9E9, 9E9]];
	VAR robtarget OpenholeUD_6630 := [[441.66, -8.7, 182.51], [-0.059999, 0.704557, 0.707063, -0.00785], [0,0,0,0], [9E9, 9E9, 9E9, 9E9, 9E9, 9E9]];
	VAR robtarget OpenholeUD_6631 := [[437.68, -8.7, 182.9], [-0.073319, 0.703295, 0.707084, 0.00563], [0,0,0,0], [9E9, 9E9, 9E9, 9E9, 9E9, 9E9]];
	VAR robtarget OpenholeUD_6632 := [[433.7, -8.7, 183.3], [-0.086454, 0.701802, 0.70685, 0.01904], [0,0,0,0], [9E9, 9E9, 9E9, 9E9, 9E9, 9E9]];
	VAR robtarget OpenholeUD_6633 := [[429.72, -8.7, 183.69], [-0.099366, 0.70009, 0.706367, 0.032338], [0,0,0,0], [9E9, 9E9, 9E9, 9E9, 9E9, 9E9]];
	VAR robtarget OpenholeUD_6634 := [[425.74, -8.7, 184.09], [-0.112021, 0.698177, 0.705642, 0.045486], [0,0,0,0], [9E9, 9E9, 9E9, 9E9, 9E9, 9E9]];
	VAR robtarget OpenholeUD_6635 := [[421.76, -8.7, 184.48], [-0.124388, 0.69608, 0.704687, 0.058446], [0,0,0,0], [9E9, 9E9, 9E9, 9E9, 9E9, 9E9]];
	VAR robtarget OpenholeUD_6636 := [[417.78, -8.7, 184.88], [-0.136442, 0.693818, 0.703515, 0.071185], [0,0,0,0], [9E9, 9E9, 9E9, 9E9, 9E9, 9E9]];
	VAR robtarget OpenholeUD_6637 := [[413.8, -8.7, 185.28], [-0.148161, 0.69141, 0.702139, 0.083674], [0,0,0,0], [9E9, 9E9, 9E9, 9E9, 9E9, 9E9]];
	VAR robtarget OpenholeUD_6638 := [[409.82, -8.7, 185.67], [-0.159529, 0.688876, 0.700575, 0.095886], [0,0,0,0], [9E9, 9E9, 9E9, 9E9, 9E9, 9E9]];
	VAR robtarget OpenholeUD_6639 := [[405.84, -8.7, 186.07], [-0.170532, 0.686235, 0.698841, 0.107801], [0,0,0,0], [9E9, 9E9, 9E9, 9E9, 9E9, 9E9]];
	VAR robtarget OpenholeUD_6640 := [[401.86, -8.7, 186.46], [-0.181163, 0.683506, 0.696953, 0.1194], [0,0,0,0], [9E9, 9E9, 9E9, 9E9, 9E9, 9E9]];
	VAR robtarget OpenholeUD_6641 := [[397.88, -8.7, 186.86], [-0.191416, 0.680706, 0.694928, 0.130669], [0,0,0,0], [9E9, 9E9, 9E9, 9E9, 9E9, 9E9]];
	VAR robtarget OpenholeUD_6642 := [[393.9, -8.7, 187.25], [-0.201289, 0.677852, 0.692784, 0.141598], [0,0,0,0], [9E9, 9E9, 9E9, 9E9, 9E9, 9E9]];
	VAR robtarget OpenholeUD_6643 := [[389.37, -8.7, 187.7], [-0.212071, 0.674556, 0.690218, 0.15362], [0,0,0,0], [9E9, 9E9, 9E9, 9E9, 9E9, 9E9]];
	VAR robtarget OpenholeUD_6644 := [[385.37, -8.7, 187.72], [-0.183051, 0.683002, 0.683002, 0.183051], [0,0,0,0], [9E9, 9E9, 9E9, 9E9, 9E9, 9E9]];
	VAR robtarget OpenholeUD_6645 := [[381.37, -8.7, 187.73], [-0.183051, 0.683002, 0.683002, 0.183051], [0,0,0,0], [9E9, 9E9, 9E9, 9E9, 9E9, 9E9]];
	VAR robtarget OpenholeUD_6646 := [[377.37, -8.7, 187.74], [-0.183051, 0.683002, 0.683002, 0.183051], [0,0,0,0], [9E9, 9E9, 9E9, 9E9, 9E9, 9E9]];
	VAR robtarget OpenholeUD_6647 := [[373.37, -8.7, 187.76], [-0.183051, 0.683002, 0.683002, 0.183051], [0,0,0,0], [9E9, 9E9, 9E9, 9E9, 9E9, 9E9]];
	VAR robtarget OpenholeUD_6648 := [[369.37, -8.7, 187.77], [-0.183051, 0.683002, 0.683002, 0.183051], [0,0,0,0], [9E9, 9E9, 9E9, 9E9, 9E9, 9E9]];
	VAR robtarget OpenholeUD_6649 := [[369.37, -8.7, 187.77], [-0.183051, 0.683002, 0.683002, 0.183051], [0,0,0,0], [9E9, 9E9, 9E9, 9E9, 9E9, 9E9]];
	VAR robtarget OpenholeUD_6650 := [[369.37, -7.5, 188.46], [-0.183051, 0.683002, 0.683002, 0.183051], [0,0,0,0], [9E9, 9E9, 9E9, 9E9, 9E9, 9E9]];
	VAR robtarget OpenholeUD_6651 := [[373.37, -7.5, 188.45], [-0.183051, 0.683002, 0.683002, 0.183051], [0,0,0,0], [9E9, 9E9, 9E9, 9E9, 9E9, 9E9]];
	VAR robtarget OpenholeUD_6652 := [[377.37, -7.5, 188.44], [-0.183051, 0.683002, 0.683002, 0.183051], [0,0,0,0], [9E9, 9E9, 9E9, 9E9, 9E9, 9E9]];
	VAR robtarget OpenholeUD_6653 := [[381.37, -7.5, 188.42], [-0.183051, 0.683002, 0.683002, 0.183051], [0,0,0,0], [9E9, 9E9, 9E9, 9E9, 9E9, 9E9]];
	VAR robtarget OpenholeUD_6654 := [[385.37, -7.5, 188.41], [-0.183051, 0.683002, 0.683002, 0.183051], [0,0,0,0], [9E9, 9E9, 9E9, 9E9, 9E9, 9E9]];
	VAR robtarget OpenholeUD_6655 := [[389.37, -7.5, 188.4], [-0.215423, 0.673493, 0.690969, 0.150204], [0,0,0,0], [9E9, 9E9, 9E9, 9E9, 9E9, 9E9]];
	VAR robtarget OpenholeUD_6656 := [[393.34, -7.5, 187.96], [-0.20606, 0.676416, 0.693186, 0.139618], [0,0,0,0], [9E9, 9E9, 9E9, 9E9, 9E9, 9E9]];
	VAR robtarget OpenholeUD_6657 := [[397.32, -7.5, 187.52], [-0.19632, 0.679307, 0.695299, 0.128685], [0,0,0,0], [9E9, 9E9, 9E9, 9E9, 9E9, 9E9]];
	VAR robtarget OpenholeUD_6658 := [[401.29, -7.5, 187.07], [-0.1862, 0.682151, 0.69729, 0.117414], [0,0,0,0], [9E9, 9E9, 9E9, 9E9, 9E9, 9E9]];
	VAR robtarget OpenholeUD_6659 := [[405.27, -7.5, 186.63], [-0.175701, 0.68493, 0.699145, 0.105815], [0,0,0,0], [9E9, 9E9, 9E9, 9E9, 9E9, 9E9]];
	VAR robtarget OpenholeUD_6660 := [[409.25, -7.5, 186.19], [-0.164826, 0.687628, 0.700844, 0.093902], [0,0,0,0], [9E9, 9E9, 9E9, 9E9, 9E9, 9E9]];
	VAR robtarget OpenholeUD_6661 := [[413.22, -7.5, 185.75], [-0.153584, 0.690226, 0.702372, 0.081692], [0,0,0,0], [9E9, 9E9, 9E9, 9E9, 9E9, 9E9]];
	VAR robtarget OpenholeUD_6662 := [[417.2, -7.5, 185.31], [-0.141984, 0.692705, 0.703712, 0.069208], [0,0,0,0], [9E9, 9E9, 9E9, 9E9, 9E9, 9E9]];
	VAR robtarget OpenholeUD_6663 := [[421.17, -7.5, 184.87], [-0.130045, 0.695046, 0.704848, 0.056474], [0,0,0,0], [9E9, 9E9, 9E9, 9E9, 9E9, 9E9]];
	VAR robtarget OpenholeUD_6664 := [[425.15, -7.5, 184.43], [-0.117784, 0.697228, 0.705766, 0.04352], [0,0,0,0], [9E9, 9E9, 9E9, 9E9, 9E9, 9E9]];
	VAR robtarget OpenholeUD_6665 := [[429.12, -7.5, 183.99], [-0.105227, 0.699233, 0.706454, 0.03038], [0,0,0,0], [9E9, 9E9, 9E9, 9E9, 9E9, 9E9]];
	VAR robtarget OpenholeUD_6666 := [[433.1, -7.5, 183.54], [-0.092403, 0.701043, 0.7069, 0.017089], [0,0,0,0], [9E9, 9E9, 9E9, 9E9, 9E9, 9E9]];
	VAR robtarget OpenholeUD_6667 := [[437.08, -7.5, 183.1], [-0.079344, 0.702641, 0.707097, 0.003688], [0,0,0,0], [9E9, 9E9, 9E9, 9E9, 9E9, 9E9]];
	VAR robtarget OpenholeUD_6668 := [[441.05, -7.5, 182.66], [-0.066088, 0.704012, 0.707039, -0.009783], [0,0,0,0], [9E9, 9E9, 9E9, 9E9, 9E9, 9E9]];
	VAR robtarget OpenholeUD_6669 := [[445.03, -7.5, 182.22], [-0.052675, 0.705142, 0.706723, -0.023281], [0,0,0,0], [9E9, 9E9, 9E9, 9E9, 9E9, 9E9]];
	VAR robtarget OpenholeUD_6670 := [[449, -7.5, 181.78], [-0.039146, 0.706022, 0.706151, -0.036761], [0,0,0,0], [9E9, 9E9, 9E9, 9E9, 9E9, 9E9]];
	VAR robtarget OpenholeUD_6671 := [[452.98, -7.5, 181.34], [-0.025547, 0.706645, 0.705324, -0.05018], [0,0,0,0], [9E9, 9E9, 9E9, 9E9, 9E9, 9E9]];
	VAR robtarget OpenholeUD_6672 := [[456.95, -7.5, 180.9], [-0.011924, 0.707006, 0.70425, -0.063494], [0,0,0,0], [9E9, 9E9, 9E9, 9E9, 9E9, 9E9]];
	VAR robtarget OpenholeUD_6673 := [[460.93, -7.5, 180.46], [0.001679, 0.707105, 0.702939, -0.076663], [0,0,0,0], [9E9, 9E9, 9E9, 9E9, 9E9, 9E9]];
	VAR robtarget OpenholeUD_6674 := [[464.9, -7.5, 180.01], [0.015216, 0.706943, 0.701401, -0.089646], [0,0,0,0], [9E9, 9E9, 9E9, 9E9, 9E9, 9E9]];
	VAR robtarget OpenholeUD_6675 := [[468.88, -7.5, 179.57], [0.028644, 0.706526, 0.699652, -0.102409], [0,0,0,0], [9E9, 9E9, 9E9, 9E9, 9E9, 9E9]];
	VAR robtarget OpenholeUD_6676 := [[472.86, -7.5, 179.13], [0.041922, 0.705863, 0.697706, -0.114919], [0,0,0,0], [9E9, 9E9, 9E9, 9E9, 9E9, 9E9]];
	VAR robtarget OpenholeUD_6677 := [[476.83, -7.5, 178.69], [0.055012, 0.704964, 0.695582, -0.127145], [0,0,0,0], [9E9, 9E9, 9E9, 9E9, 9E9, 9E9]];
	VAR robtarget OpenholeUD_6678 := [[480.81, -7.5, 178.25], [0.067878, 0.703841, 0.693297, -0.139065], [0,0,0,0], [9E9, 9E9, 9E9, 9E9, 9E9, 9E9]];
	VAR robtarget OpenholeUD_6679 := [[484.78, -7.5, 177.81], [0.080491, 0.702511, 0.690871, -0.150656], [0,0,0,0], [9E9, 9E9, 9E9, 9E9, 9E9, 9E9]];
	VAR robtarget OpenholeUD_6680 := [[488.76, -7.5, 177.37], [0.092824, 0.700988, 0.688322, -0.161904], [0,0,0,0], [9E9, 9E9, 9E9, 9E9, 9E9, 9E9]];
	VAR robtarget OpenholeUD_6681 := [[492.73, -7.5, 176.93], [0.104854, 0.699289, 0.685669, -0.172794], [0,0,0,0], [9E9, 9E9, 9E9, 9E9, 9E9, 9E9]];
	VAR robtarget OpenholeUD_6682 := [[496.71, -7.5, 176.49], [0.116563, 0.697433, 0.68293, -0.18332], [0,0,0,0], [9E9, 9E9, 9E9, 9E9, 9E9, 9E9]];
	VAR robtarget OpenholeUD_6683 := [[500.68, -7.5, 176.04], [0.127937, 0.695437, 0.680123, -0.193475], [0,0,0,0], [9E9, 9E9, 9E9, 9E9, 9E9, 9E9]];
	VAR robtarget OpenholeUD_6684 := [[504.66, -7.5, 175.6], [0.138965, 0.693317, 0.677264, -0.203259], [0,0,0,0], [9E9, 9E9, 9E9, 9E9, 9E9, 9E9]];
	VAR robtarget OpenholeUD_6685 := [[509.33, -7.5, 175.08], [0.183051, 0.683002, 0.683002, -0.183051], [0,0,0,0], [9E9, 9E9, 9E9, 9E9, 9E9, 9E9]];
	VAR robtarget OpenholeUD_6686 := [[513.33, -7.5, 175.07], [0.183051, 0.683002, 0.683002, -0.183051], [0,0,0,0], [9E9, 9E9, 9E9, 9E9, 9E9, 9E9]];
	VAR robtarget OpenholeUD_6687 := [[517.33, -7.5, 175.06], [0.183051, 0.683002, 0.683002, -0.183051], [0,0,0,0], [9E9, 9E9, 9E9, 9E9, 9E9, 9E9]];
	VAR robtarget OpenholeUD_6688 := [[521.33, -7.5, 175.05], [0.183051, 0.683002, 0.683002, -0.183051], [0,0,0,0], [9E9, 9E9, 9E9, 9E9, 9E9, 9E9]];
	VAR robtarget OpenholeUD_6689 := [[525.33, -7.5, 175.03], [0.183051, 0.683002, 0.683002, -0.183051], [0,0,0,0], [9E9, 9E9, 9E9, 9E9, 9E9, 9E9]];
	VAR robtarget OpenholeUD_6690 := [[529.33, -7.5, 175.02], [0.183051, 0.683002, 0.683002, -0.183051], [0,0,0,0], [9E9, 9E9, 9E9, 9E9, 9E9, 9E9]];
	VAR robtarget OpenholeUD_6691 := [[529.33, -7.5, 175.02], [0.183051, 0.683002, 0.683002, -0.183051], [0,0,0,0], [9E9, 9E9, 9E9, 9E9, 9E9, 9E9]];
	VAR robtarget OpenholeUD_6692 := [[529.32, -6.3, 174.33], [0.183051, 0.683002, 0.683002, -0.183051], [0,0,0,0], [9E9, 9E9, 9E9, 9E9, 9E9, 9E9]];
	VAR robtarget OpenholeUD_6693 := [[525.32, -6.3, 174.34], [0.183051, 0.683002, 0.683002, -0.183051], [0,0,0,0], [9E9, 9E9, 9E9, 9E9, 9E9, 9E9]];
	VAR robtarget OpenholeUD_6694 := [[521.32, -6.3, 174.35], [0.183051, 0.683002, 0.683002, -0.183051], [0,0,0,0], [9E9, 9E9, 9E9, 9E9, 9E9, 9E9]];
	VAR robtarget OpenholeUD_6695 := [[517.32, -6.3, 174.37], [0.183051, 0.683002, 0.683002, -0.183051], [0,0,0,0], [9E9, 9E9, 9E9, 9E9, 9E9, 9E9]];
	VAR robtarget OpenholeUD_6696 := [[513.32, -6.3, 174.38], [0.183051, 0.683002, 0.683002, -0.183051], [0,0,0,0], [9E9, 9E9, 9E9, 9E9, 9E9, 9E9]];
	VAR robtarget OpenholeUD_6697 := [[509.32, -6.3, 174.39], [0.183051, 0.683002, 0.683002, -0.183051], [0,0,0,0], [9E9, 9E9, 9E9, 9E9, 9E9, 9E9]];
	VAR robtarget OpenholeUD_6698 := [[505.35, -6.3, 174.88], [0.137356, 0.693638, 0.675722, -0.208327], [0,0,0,0], [9E9, 9E9, 9E9, 9E9, 9E9, 9E9]];
	VAR robtarget OpenholeUD_6699 := [[501.38, -6.3, 175.36], [0.126339, 0.695729, 0.678619, -0.198688], [0,0,0,0], [9E9, 9E9, 9E9, 9E9, 9E9, 9E9]];
	VAR robtarget OpenholeUD_6700 := [[497.41, -6.3, 175.85], [0.114977, 0.697696, 0.68147, -0.188677], [0,0,0,0], [9E9, 9E9, 9E9, 9E9, 9E9, 9E9]];
	VAR robtarget OpenholeUD_6701 := [[493.44, -6.3, 176.34], [0.103281, 0.699523, 0.68426, -0.178294], [0,0,0,0], [9E9, 9E9, 9E9, 9E9, 9E9, 9E9]];
	VAR robtarget OpenholeUD_6702 := [[489.47, -6.3, 176.82], [0.091265, 0.701192, 0.686971, -0.167543], [0,0,0,0], [9E9, 9E9, 9E9, 9E9, 9E9, 9E9]];
	VAR robtarget OpenholeUD_6703 := [[485.5, -6.3, 177.31], [0.078947, 0.702686, 0.689586, -0.156432], [0,0,0,0], [9E9, 9E9, 9E9, 9E9, 9E9, 9E9]];
	VAR robtarget OpenholeUD_6704 := [[481.53, -6.3, 177.8], [0.066349, 0.703987, 0.692086, -0.144971], [0,0,0,0], [9E9, 9E9, 9E9, 9E9, 9E9, 9E9]];
	VAR robtarget OpenholeUD_6705 := [[477.56, -6.3, 178.28], [0.053498, 0.70508, 0.694452, -0.133176], [0,0,0,0], [9E9, 9E9, 9E9, 9E9, 9E9, 9E9]];
	VAR robtarget OpenholeUD_6706 := [[473.59, -6.3, 178.77], [0.040424, 0.70595, 0.696666, -0.121065], [0,0,0,0], [9E9, 9E9, 9E9, 9E9, 9E9, 9E9]];
	VAR robtarget OpenholeUD_6707 := [[469.62, -6.3, 179.26], [0.027162, 0.706585, 0.698708, -0.108663], [0,0,0,0], [9E9, 9E9, 9E9, 9E9, 9E9, 9E9]];
	VAR robtarget OpenholeUD_6708 := [[465.65, -6.3, 179.74], [0.013748, 0.706973, 0.70056, -0.095996], [0,0,0,0], [9E9, 9E9, 9E9, 9E9, 9E9, 9E9]];
	VAR robtarget OpenholeUD_6709 := [[461.68, -6.3, 180.23], [0.000225, 0.707107, 0.702207, -0.083097], [0,0,0,0], [9E9, 9E9, 9E9, 9E9, 9E9, 9E9]];
	VAR robtarget OpenholeUD_6710 := [[457.71, -6.3, 180.72], [-0.013365, 0.70698, 0.703634, -0.069999], [0,0,0,0], [9E9, 9E9, 9E9, 9E9, 9E9, 9E9]];
	VAR robtarget OpenholeUD_6711 := [[453.74, -6.3, 181.2], [-0.026978, 0.706592, 0.704826, -0.056742], [0,0,0,0], [9E9, 9E9, 9E9, 9E9, 9E9, 9E9]];
	VAR robtarget OpenholeUD_6712 := [[449.77, -6.3, 181.69], [-0.040567, 0.705942, 0.705776, -0.043365], [0,0,0,0], [9E9, 9E9, 9E9, 9E9, 9E9, 9E9]];
	VAR robtarget OpenholeUD_6713 := [[445.8, -6.3, 182.18], [-0.054088, 0.705035, 0.706474, -0.029913], [0,0,0,0], [9E9, 9E9, 9E9, 9E9, 9E9, 9E9]];
	VAR robtarget OpenholeUD_6714 := [[441.83, -6.3, 182.66], [-0.067495, 0.703878, 0.706916, -0.016427], [0,0,0,0], [9E9, 9E9, 9E9, 9E9, 9E9, 9E9]];
	VAR robtarget OpenholeUD_6715 := [[437.86, -6.3, 183.15], [-0.080746, 0.702481, 0.707101, -0.002952], [0,0,0,0], [9E9, 9E9, 9E9, 9E9, 9E9, 9E9]];
	VAR robtarget OpenholeUD_6716 := [[433.89, -6.3, 183.64], [-0.093801, 0.700858, 0.707029, 0.010469], [0,0,0,0], [9E9, 9E9, 9E9, 9E9, 9E9, 9E9]];
	VAR robtarget OpenholeUD_6717 := [[429.92, -6.3, 184.12], [-0.106623, 0.699022, 0.706706, 0.023794], [0,0,0,0], [9E9, 9E9, 9E9, 9E9, 9E9, 9E9]];
	VAR robtarget OpenholeUD_6718 := [[425.95, -6.3, 184.61], [-0.119179, 0.696991, 0.706139, 0.036982], [0,0,0,0], [9E9, 9E9, 9E9, 9E9, 9E9, 9E9]];
	VAR robtarget OpenholeUD_6719 := [[421.98, -6.3, 185.1], [-0.131439, 0.694783, 0.705337, 0.049998], [0,0,0,0], [9E9, 9E9, 9E9, 9E9, 9E9, 9E9]];
	VAR robtarget OpenholeUD_6720 := [[418.01, -6.3, 185.58], [-0.14338, 0.692418, 0.704312, 0.062805], [0,0,0,0], [9E9, 9E9, 9E9, 9E9, 9E9, 9E9]];
	VAR robtarget OpenholeUD_6721 := [[414.04, -6.3, 186.07], [-0.154979, 0.689914, 0.703078, 0.075374], [0,0,0,0], [9E9, 9E9, 9E9, 9E9, 9E9, 9E9]];
	VAR robtarget OpenholeUD_6722 := [[410.07, -6.3, 186.55], [-0.166223, 0.687292, 0.70165, 0.087679], [0,0,0,0], [9E9, 9E9, 9E9, 9E9, 9E9, 9E9]];
	VAR robtarget OpenholeUD_6723 := [[406.1, -6.3, 187.04], [-0.177098, 0.68457, 0.700044, 0.099695], [0,0,0,0], [9E9, 9E9, 9E9, 9E9, 9E9, 9E9]];
	VAR robtarget OpenholeUD_6724 := [[402.13, -6.3, 187.53], [-0.187598, 0.681768, 0.698276, 0.111404], [0,0,0,0], [9E9, 9E9, 9E9, 9E9, 9E9, 9E9]];
	VAR robtarget OpenholeUD_6725 := [[398.16, -6.3, 188.01], [-0.197718, 0.678902, 0.696364, 0.122791], [0,0,0,0], [9E9, 9E9, 9E9, 9E9, 9E9, 9E9]];
	VAR robtarget OpenholeUD_6726 := [[394.19, -6.3, 188.5], [-0.207457, 0.675989, 0.694324, 0.133844], [0,0,0,0], [9E9, 9E9, 9E9, 9E9, 9E9, 9E9]];
	VAR robtarget OpenholeUD_6727 := [[389.37, -6.3, 189.09], [-0.218763, 0.672416, 0.691702, 0.146792], [0,0,0,0], [9E9, 9E9, 9E9, 9E9, 9E9, 9E9]];
	VAR robtarget OpenholeUD_6728 := [[385.37, -6.3, 189.1], [-0.183051, 0.683002, 0.683002, 0.183051], [0,0,0,0], [9E9, 9E9, 9E9, 9E9, 9E9, 9E9]];
	VAR robtarget OpenholeUD_6729 := [[381.37, -6.3, 189.12], [-0.183051, 0.683002, 0.683002, 0.183051], [0,0,0,0], [9E9, 9E9, 9E9, 9E9, 9E9, 9E9]];
	VAR robtarget OpenholeUD_6730 := [[377.37, -6.3, 189.13], [-0.183051, 0.683002, 0.683002, 0.183051], [0,0,0,0], [9E9, 9E9, 9E9, 9E9, 9E9, 9E9]];
	VAR robtarget OpenholeUD_6731 := [[373.37, -6.3, 189.14], [-0.183051, 0.683002, 0.683002, 0.183051], [0,0,0,0], [9E9, 9E9, 9E9, 9E9, 9E9, 9E9]];
	VAR robtarget OpenholeUD_6732 := [[369.37, -6.3, 189.15], [-0.183051, 0.683002, 0.683002, 0.183051], [0,0,0,0], [9E9, 9E9, 9E9, 9E9, 9E9, 9E9]];
	VAR robtarget OpenholeUD_6733 := [[369.37, -6.3, 189.15], [-0.183051, 0.683002, 0.683002, 0.183051], [0,0,0,0], [9E9, 9E9, 9E9, 9E9, 9E9, 9E9]];
	VAR robtarget OpenholeUD_6734 := [[369.37, -5.1, 189.85], [-0.183051, 0.683002, 0.683002, 0.183051], [0,0,0,0], [9E9, 9E9, 9E9, 9E9, 9E9, 9E9]];
	VAR robtarget OpenholeUD_6735 := [[373.37, -5.1, 189.83], [-0.183051, 0.683002, 0.683002, 0.183051], [0,0,0,0], [9E9, 9E9, 9E9, 9E9, 9E9, 9E9]];
	VAR robtarget OpenholeUD_6736 := [[377.37, -5.1, 189.82], [-0.183051, 0.683002, 0.683002, 0.183051], [0,0,0,0], [9E9, 9E9, 9E9, 9E9, 9E9, 9E9]];
	VAR robtarget OpenholeUD_6737 := [[381.37, -5.1, 189.81], [-0.183051, 0.683002, 0.683002, 0.183051], [0,0,0,0], [9E9, 9E9, 9E9, 9E9, 9E9, 9E9]];
	VAR robtarget OpenholeUD_6738 := [[385.37, -5.1, 189.8], [-0.183051, 0.683002, 0.683002, 0.183051], [0,0,0,0], [9E9, 9E9, 9E9, 9E9, 9E9, 9E9]];
	VAR robtarget OpenholeUD_6739 := [[389.37, -5.1, 189.78], [-0.22209, 0.671324, 0.692417, 0.143383], [0,0,0,0], [9E9, 9E9, 9E9, 9E9, 9E9, 9E9]];
	VAR robtarget OpenholeUD_6740 := [[393.34, -5.1, 189.25], [-0.212891, 0.674298, 0.694544, 0.132696], [0,0,0,0], [9E9, 9E9, 9E9, 9E9, 9E9, 9E9]];
	VAR robtarget OpenholeUD_6741 := [[397.3, -5.1, 188.72], [-0.203315, 0.677247, 0.696561, 0.121668], [0,0,0,0], [9E9, 9E9, 9E9, 9E9, 9E9, 9E9]];
	VAR robtarget OpenholeUD_6742 := [[401.27, -5.1, 188.19], [-0.193358, 0.680156, 0.69845, 0.110308], [0,0,0,0], [9E9, 9E9, 9E9, 9E9, 9E9, 9E9]];
	VAR robtarget OpenholeUD_6743 := [[405.23, -5.1, 187.66], [-0.183021, 0.683011, 0.700195, 0.098625], [0,0,0,0], [9E9, 9E9, 9E9, 9E9, 9E9, 9E9]];
	VAR robtarget OpenholeUD_6744 := [[409.2, -5.1, 187.13], [-0.172305, 0.685792, 0.701779, 0.086636], [0,0,0,0], [9E9, 9E9, 9E9, 9E9, 9E9, 9E9]];
	VAR robtarget OpenholeUD_6745 := [[413.16, -5.1, 186.59], [-0.161217, 0.688483, 0.703186, 0.074359], [0,0,0,0], [9E9, 9E9, 9E9, 9E9, 9E9, 9E9]];
	VAR robtarget OpenholeUD_6746 := [[417.12, -5.1, 186.06], [-0.149767, 0.691064, 0.7044, 0.061816], [0,0,0,0], [9E9, 9E9, 9E9, 9E9, 9E9, 9E9]];
	VAR robtarget OpenholeUD_6747 := [[421.09, -5.1, 185.53], [-0.137971, 0.693516, 0.705405, 0.049034], [0,0,0,0], [9E9, 9E9, 9E9, 9E9, 9E9, 9E9]];
	VAR robtarget OpenholeUD_6748 := [[425.05, -5.1, 185], [-0.125845, 0.695818, 0.706188, 0.036043], [0,0,0,0], [9E9, 9E9, 9E9, 9E9, 9E9, 9E9]];
	VAR robtarget OpenholeUD_6749 := [[429.02, -5.1, 184.47], [-0.113414, 0.697952, 0.706737, 0.022876], [0,0,0,0], [9E9, 9E9, 9E9, 9E9, 9E9, 9E9]];
	VAR robtarget OpenholeUD_6750 := [[432.98, -5.1, 183.94], [-0.100704, 0.699899, 0.707042, 0.009571], [0,0,0,0], [9E9, 9E9, 9E9, 9E9, 9E9, 9E9]];
	VAR robtarget OpenholeUD_6751 := [[436.95, -5.1, 183.4], [-0.087748, 0.701641, 0.707096, -0.003832], [0,0,0,0], [9E9, 9E9, 9E9, 9E9, 9E9, 9E9]];
	VAR robtarget OpenholeUD_6752 := [[440.91, -5.1, 182.87], [-0.074581, 0.703163, 0.706895, -0.017294], [0,0,0,0], [9E9, 9E9, 9E9, 9E9, 9E9, 9E9]];
	VAR robtarget OpenholeUD_6753 := [[444.88, -5.1, 182.34], [-0.061242, 0.70445, 0.706437, -0.030769], [0,0,0,0], [9E9, 9E9, 9E9, 9E9, 9E9, 9E9]];
	VAR robtarget OpenholeUD_6754 := [[448.84, -5.1, 181.81], [-0.047773, 0.705491, 0.705723, -0.044214], [0,0,0,0], [9E9, 9E9, 9E9, 9E9, 9E9, 9E9]];
	VAR robtarget OpenholeUD_6755 := [[452.8, -5.1, 181.28], [-0.034218, 0.706278, 0.704758, -0.057586], [0,0,0,0], [9E9, 9E9, 9E9, 9E9, 9E9, 9E9]];
	VAR robtarget OpenholeUD_6756 := [[456.77, -5.1, 180.75], [-0.020621, 0.706806, 0.703549, -0.070843], [0,0,0,0], [9E9, 9E9, 9E9, 9E9, 9E9, 9E9]];
	VAR robtarget OpenholeUD_6757 := [[460.73, -5.1, 180.21], [-0.007029, 0.707072, 0.702107, -0.083943], [0,0,0,0], [9E9, 9E9, 9E9, 9E9, 9E9, 9E9]];
	VAR robtarget OpenholeUD_6758 := [[464.7, -5.1, 179.68], [0.006514, 0.707077, 0.700443, -0.096847], [0,0,0,0], [9E9, 9E9, 9E9, 9E9, 9E9, 9E9]];
	VAR robtarget OpenholeUD_6759 := [[468.66, -5.1, 179.15], [0.019965, 0.706825, 0.698574, -0.109522], [0,0,0,0], [9E9, 9E9, 9E9, 9E9, 9E9, 9E9]];
	VAR robtarget OpenholeUD_6760 := [[472.63, -5.1, 178.62], [0.03328, 0.706323, 0.696514, -0.121934], [0,0,0,0], [9E9, 9E9, 9E9, 9E9, 9E9, 9E9]];
	VAR robtarget OpenholeUD_6761 := [[476.59, -5.1, 178.09], [0.046423, 0.705581, 0.694283, -0.134057], [0,0,0,0], [9E9, 9E9, 9E9, 9E9, 9E9, 9E9]];
	VAR robtarget OpenholeUD_6762 := [[480.56, -5.1, 177.56], [0.059356, 0.704611, 0.691898, -0.145865], [0,0,0,0], [9E9, 9E9, 9E9, 9E9, 9E9, 9E9]];
	VAR robtarget OpenholeUD_6763 := [[484.52, -5.1, 177.02], [0.072049, 0.703427, 0.689379, -0.157341], [0,0,0,0], [9E9, 9E9, 9E9, 9E9, 9E9, 9E9]];
	VAR robtarget OpenholeUD_6764 := [[488.49, -5.1, 176.49], [0.084473, 0.702043, 0.686745, -0.168467], [0,0,0,0], [9E9, 9E9, 9E9, 9E9, 9E9, 9E9]];
	VAR robtarget OpenholeUD_6765 := [[492.45, -5.1, 175.96], [0.096605, 0.700477, 0.684014, -0.179233], [0,0,0,0], [9E9, 9E9, 9E9, 9E9, 9E9, 9E9]];
	VAR robtarget OpenholeUD_6766 := [[496.41, -5.1, 175.43], [0.108426, 0.698744, 0.681205, -0.189631], [0,0,0,0], [9E9, 9E9, 9E9, 9E9, 9E9, 9E9]];
	VAR robtarget OpenholeUD_6767 := [[500.38, -5.1, 174.9], [0.119919, 0.696864, 0.678334, -0.199657], [0,0,0,0], [9E9, 9E9, 9E9, 9E9, 9E9, 9E9]];
	VAR robtarget OpenholeUD_6768 := [[504.34, -5.1, 174.37], [0.131072, 0.694853, 0.675418, -0.20931], [0,0,0,0], [9E9, 9E9, 9E9, 9E9, 9E9, 9E9]];
	VAR robtarget OpenholeUD_6769 := [[509.32, -5.1, 173.7], [0.183051, 0.683002, 0.683002, -0.183051], [0,0,0,0], [9E9, 9E9, 9E9, 9E9, 9E9, 9E9]];
	VAR robtarget OpenholeUD_6770 := [[513.32, -5.1, 173.69], [0.183051, 0.683002, 0.683002, -0.183051], [0,0,0,0], [9E9, 9E9, 9E9, 9E9, 9E9, 9E9]];
	VAR robtarget OpenholeUD_6771 := [[517.32, -5.1, 173.67], [0.183051, 0.683002, 0.683002, -0.183051], [0,0,0,0], [9E9, 9E9, 9E9, 9E9, 9E9, 9E9]];
	VAR robtarget OpenholeUD_6772 := [[521.32, -5.1, 173.66], [0.183051, 0.683002, 0.683002, -0.183051], [0,0,0,0], [9E9, 9E9, 9E9, 9E9, 9E9, 9E9]];
	VAR robtarget OpenholeUD_6773 := [[525.32, -5.1, 173.65], [0.183051, 0.683002, 0.683002, -0.183051], [0,0,0,0], [9E9, 9E9, 9E9, 9E9, 9E9, 9E9]];
	VAR robtarget OpenholeUD_6774 := [[529.32, -5.1, 173.64], [0.183051, 0.683002, 0.683002, -0.183051], [0,0,0,0], [9E9, 9E9, 9E9, 9E9, 9E9, 9E9]];
	VAR robtarget OpenholeUD_6775 := [[529.32, -5.1, 173.64], [0.183051, 0.683002, 0.683002, -0.183051], [0,0,0,0], [9E9, 9E9, 9E9, 9E9, 9E9, 9E9]];
	VAR robtarget OpenholeUD_6776 := [[529.32, -3.9, 172.94], [0.183051, 0.683002, 0.683002, -0.183051], [0,0,0,0], [9E9, 9E9, 9E9, 9E9, 9E9, 9E9]];
	VAR robtarget OpenholeUD_6777 := [[525.32, -3.9, 172.96], [0.183051, 0.683002, 0.683002, -0.183051], [0,0,0,0], [9E9, 9E9, 9E9, 9E9, 9E9, 9E9]];
	VAR robtarget OpenholeUD_6778 := [[521.32, -3.9, 172.97], [0.183051, 0.683002, 0.683002, -0.183051], [0,0,0,0], [9E9, 9E9, 9E9, 9E9, 9E9, 9E9]];
	VAR robtarget OpenholeUD_6779 := [[517.32, -3.9, 172.98], [0.183051, 0.683002, 0.683002, -0.183051], [0,0,0,0], [9E9, 9E9, 9E9, 9E9, 9E9, 9E9]];
	VAR robtarget OpenholeUD_6780 := [[513.32, -3.9, 172.99], [0.183051, 0.683002, 0.683002, -0.183051], [0,0,0,0], [9E9, 9E9, 9E9, 9E9, 9E9, 9E9]];
	VAR robtarget OpenholeUD_6781 := [[509.32, -3.9, 173.01], [0.183051, 0.683002, 0.683002, -0.183051], [0,0,0,0], [9E9, 9E9, 9E9, 9E9, 9E9, 9E9]];
	VAR robtarget OpenholeUD_6782 := [[505.36, -3.9, 173.58], [0.130393, 0.69498, 0.673595, -0.215104], [0,0,0,0], [9E9, 9E9, 9E9, 9E9, 9E9, 9E9]];
	VAR robtarget OpenholeUD_6783 := [[501.4, -3.9, 174.16], [0.119281, 0.696973, 0.676548, -0.205628], [0,0,0,0], [9E9, 9E9, 9E9, 9E9, 9E9, 9E9]];
	VAR robtarget OpenholeUD_6784 := [[497.45, -3.9, 174.74], [0.107831, 0.698836, 0.679464, -0.195779], [0,0,0,0], [9E9, 9E9, 9E9, 9E9, 9E9, 9E9]];
	VAR robtarget OpenholeUD_6785 := [[493.49, -3.9, 175.31], [0.096054, 0.700552, 0.682326, -0.185556], [0,0,0,0], [9E9, 9E9, 9E9, 9E9, 9E9, 9E9]];
	VAR robtarget OpenholeUD_6786 := [[489.53, -3.9, 175.89], [0.083964, 0.702104, 0.685119, -0.174963], [0,0,0,0], [9E9, 9E9, 9E9, 9E9, 9E9, 9E9]];
	VAR robtarget OpenholeUD_6787 := [[485.57, -3.9, 176.47], [0.071581, 0.703474, 0.687824, -0.164005], [0,0,0,0], [9E9, 9E9, 9E9, 9E9, 9E9, 9E9]];
	VAR robtarget OpenholeUD_6788 := [[481.61, -3.9, 177.04], [0.058928, 0.704647, 0.690424, -0.152693], [0,0,0,0], [9E9, 9E9, 9E9, 9E9, 9E9, 9E9]];
	VAR robtarget OpenholeUD_6789 := [[477.65, -3.9, 177.62], [0.046032, 0.705607, 0.692898, -0.14104], [0,0,0,0], [9E9, 9E9, 9E9, 9E9, 9E9, 9E9]];
	VAR robtarget OpenholeUD_6790 := [[473.7, -3.9, 178.19], [0.032924, 0.70634, 0.695228, -0.129064], [0,0,0,0], [9E9, 9E9, 9E9, 9E9, 9E9, 9E9]];
	VAR robtarget OpenholeUD_6791 := [[469.74, -3.9, 178.77], [0.01964, 0.706834, 0.697396, -0.116787], [0,0,0,0], [9E9, 9E9, 9E9, 9E9, 9E9, 9E9]];
	VAR robtarget OpenholeUD_6792 := [[465.78, -3.9, 179.35], [0.006216, 0.707079, 0.699382, -0.104235], [0,0,0,0], [9E9, 9E9, 9E9, 9E9, 9E9, 9E9]];
	VAR robtarget OpenholeUD_6793 := [[461.82, -3.9, 179.92], [-0.007305, 0.707069, 0.70117, -0.091438], [0,0,0,0], [9E9, 9E9, 9E9, 9E9, 9E9, 9E9]];
	VAR robtarget OpenholeUD_6794 := [[457.86, -3.9, 180.5], [-0.02088, 0.706798, 0.702744, -0.078431], [0,0,0,0], [9E9, 9E9, 9E9, 9E9, 9E9, 9E9]];
	VAR robtarget OpenholeUD_6795 := [[453.91, -3.9, 181.08], [-0.034465, 0.706266, 0.70409, -0.065251], [0,0,0,0], [9E9, 9E9, 9E9, 9E9, 9E9, 9E9]];
	VAR robtarget OpenholeUD_6796 := [[449.95, -3.9, 181.65], [-0.048015, 0.705475, 0.705197, -0.051936], [0,0,0,0], [9E9, 9E9, 9E9, 9E9, 9E9, 9E9]];
	VAR robtarget OpenholeUD_6797 := [[445.99, -3.9, 182.23], [-0.061483, 0.704429, 0.706056, -0.03853], [0,0,0,0], [9E9, 9E9, 9E9, 9E9, 9E9, 9E9]];
	VAR robtarget OpenholeUD_6798 := [[442.03, -3.9, 182.81], [-0.074827, 0.703136, 0.706662, -0.025075], [0,0,0,0], [9E9, 9E9, 9E9, 9E9, 9E9, 9E9]];
	VAR robtarget OpenholeUD_6799 := [[438.07, -3.9, 183.38], [-0.088004, 0.701609, 0.707011, -0.011615], [0,0,0,0], [9E9, 9E9, 9E9, 9E9, 9E9, 9E9]];
	VAR robtarget OpenholeUD_6800 := [[434.11, -3.9, 183.96], [-0.100975, 0.69986, 0.707104, 0.001807], [0,0,0,0], [9E9, 9E9, 9E9, 9E9, 9E9, 9E9]];
	VAR robtarget OpenholeUD_6801 := [[430.16, -3.9, 184.54], [-0.113704, 0.697905, 0.706945, 0.015148], [0,0,0,0], [9E9, 9E9, 9E9, 9E9, 9E9, 9E9]];
	VAR robtarget OpenholeUD_6802 := [[426.2, -3.9, 185.11], [-0.126159, 0.695761, 0.706537, 0.028368], [0,0,0,0], [9E9, 9E9, 9E9, 9E9, 9E9, 9E9]];
	VAR robtarget OpenholeUD_6803 := [[422.24, -3.9, 185.69], [-0.138311, 0.693448, 0.705892, 0.04143], [0,0,0,0], [9E9, 9E9, 9E9, 9E9, 9E9, 9E9]];
	VAR robtarget OpenholeUD_6804 := [[418.28, -3.9, 186.27], [-0.150136, 0.690984, 0.705019, 0.054298], [0,0,0,0], [9E9, 9E9, 9E9, 9E9, 9E9, 9E9]];
	VAR robtarget OpenholeUD_6805 := [[414.32, -3.9, 186.84], [-0.161617, 0.688389, 0.703931, 0.06694], [0,0,0,0], [9E9, 9E9, 9E9, 9E9, 9E9, 9E9]];
	VAR robtarget OpenholeUD_6806 := [[410.36, -3.9, 187.42], [-0.172736, 0.685684, 0.702643, 0.079329], [0,0,0,0], [9E9, 9E9, 9E9, 9E9, 9E9, 9E9]];
	VAR robtarget OpenholeUD_6807 := [[406.41, -3.9, 188], [-0.183485, 0.682886, 0.70117, 0.09144], [0,0,0,0], [9E9, 9E9, 9E9, 9E9, 9E9, 9E9]];
	VAR robtarget OpenholeUD_6808 := [[402.45, -3.9, 188.57], [-0.193856, 0.680015, 0.699527, 0.103254], [0,0,0,0], [9E9, 9E9, 9E9, 9E9, 9E9, 9E9]];
	VAR robtarget OpenholeUD_6809 := [[398.49, -3.9, 189.15], [-0.203845, 0.677087, 0.697733, 0.114754], [0,0,0,0], [9E9, 9E9, 9E9, 9E9, 9E9, 9E9]];
	VAR robtarget OpenholeUD_6810 := [[394.53, -3.9, 189.73], [-0.213453, 0.67412, 0.695803, 0.125927], [0,0,0,0], [9E9, 9E9, 9E9, 9E9, 9E9, 9E9]];
	VAR robtarget OpenholeUD_6811 := [[389.37, -3.9, 190.48], [-0.225404, 0.670219, 0.693113, 0.139979], [0,0,0,0], [9E9, 9E9, 9E9, 9E9, 9E9, 9E9]];
	VAR robtarget OpenholeUD_6812 := [[385.37, -3.9, 190.49], [-0.183051, 0.683002, 0.683002, 0.183051], [0,0,0,0], [9E9, 9E9, 9E9, 9E9, 9E9, 9E9]];
	VAR robtarget OpenholeUD_6813 := [[381.37, -3.9, 190.5], [-0.183051, 0.683002, 0.683002, 0.183051], [0,0,0,0], [9E9, 9E9, 9E9, 9E9, 9E9, 9E9]];
	VAR robtarget OpenholeUD_6814 := [[377.37, -3.9, 190.51], [-0.183051, 0.683002, 0.683002, 0.183051], [0,0,0,0], [9E9, 9E9, 9E9, 9E9, 9E9, 9E9]];
	VAR robtarget OpenholeUD_6815 := [[373.37, -3.9, 190.53], [-0.183051, 0.683002, 0.683002, 0.183051], [0,0,0,0], [9E9, 9E9, 9E9, 9E9, 9E9, 9E9]];
	VAR robtarget OpenholeUD_6816 := [[369.37, -3.9, 190.54], [-0.183051, 0.683002, 0.683002, 0.183051], [0,0,0,0], [9E9, 9E9, 9E9, 9E9, 9E9, 9E9]];
	VAR robtarget OpenholeUD_6817 := [[369.37, -3.9, 190.54], [-0.183051, 0.683002, 0.683002, 0.183051], [0,0,0,0], [9E9, 9E9, 9E9, 9E9, 9E9, 9E9]];
	VAR robtarget OpenholeUD_6818 := [[369.38, -2.7, 191.23], [-0.183051, 0.683002, 0.683002, 0.183051], [0,0,0,0], [9E9, 9E9, 9E9, 9E9, 9E9, 9E9]];
	VAR robtarget OpenholeUD_6819 := [[373.38, -2.7, 191.22], [-0.183051, 0.683002, 0.683002, 0.183051], [0,0,0,0], [9E9, 9E9, 9E9, 9E9, 9E9, 9E9]];
	VAR robtarget OpenholeUD_6820 := [[377.38, -2.7, 191.21], [-0.183051, 0.683002, 0.683002, 0.183051], [0,0,0,0], [9E9, 9E9, 9E9, 9E9, 9E9, 9E9]];
	VAR robtarget OpenholeUD_6821 := [[381.38, -2.7, 191.2], [-0.183051, 0.683002, 0.683002, 0.183051], [0,0,0,0], [9E9, 9E9, 9E9, 9E9, 9E9, 9E9]];
	VAR robtarget OpenholeUD_6822 := [[385.38, -2.7, 191.18], [-0.183051, 0.683002, 0.683002, 0.183051], [0,0,0,0], [9E9, 9E9, 9E9, 9E9, 9E9, 9E9]];
	VAR robtarget OpenholeUD_6823 := [[389.38, -2.7, 191.17], [-0.228698, 0.669102, 0.693793, 0.136571], [0,0,0,0], [9E9, 9E9, 9E9, 9E9, 9E9, 9E9]];
	VAR robtarget OpenholeUD_6824 := [[393.33, -2.7, 190.55], [-0.219671, 0.672119, 0.695826, 0.125801], [0,0,0,0], [9E9, 9E9, 9E9, 9E9, 9E9, 9E9]];
	VAR robtarget OpenholeUD_6825 := [[397.28, -2.7, 189.93], [-0.210262, 0.675122, 0.697744, 0.114686], [0,0,0,0], [9E9, 9E9, 9E9, 9E9, 9E9, 9E9]];
	VAR robtarget OpenholeUD_6826 := [[401.23, -2.7, 189.31], [-0.200472, 0.678094, 0.699529, 0.103245], [0,0,0,0], [9E9, 9E9, 9E9, 9E9, 9E9, 9E9]];
	VAR robtarget OpenholeUD_6827 := [[405.18, -2.7, 188.68], [-0.1903, 0.681018, 0.701163, 0.091489], [0,0,0,0], [9E9, 9E9, 9E9, 9E9, 9E9, 9E9]];
	VAR robtarget OpenholeUD_6828 := [[409.13, -2.7, 188.06], [-0.179748, 0.683879, 0.702631, 0.079434], [0,0,0,0], [9E9, 9E9, 9E9, 9E9, 9E9, 9E9]];
	VAR robtarget OpenholeUD_6829 := [[413.09, -2.7, 187.44], [-0.16882, 0.686658, 0.703916, 0.067099], [0,0,0,0], [9E9, 9E9, 9E9, 9E9, 9E9, 9E9]];
	VAR robtarget OpenholeUD_6830 := [[417.04, -2.7, 186.82], [-0.157526, 0.689337, 0.705003, 0.054508], [0,0,0,0], [9E9, 9E9, 9E9, 9E9, 9E9, 9E9]];
	VAR robtarget OpenholeUD_6831 := [[420.99, -2.7, 186.2], [-0.145879, 0.691895, 0.705877, 0.041688], [0,0,0,0], [9E9, 9E9, 9E9, 9E9, 9E9, 9E9]];
	VAR robtarget OpenholeUD_6832 := [[424.94, -2.7, 185.58], [-0.133895, 0.694314, 0.706525, 0.028669], [0,0,0,0], [9E9, 9E9, 9E9, 9E9, 9E9, 9E9]];
	VAR robtarget OpenholeUD_6833 := [[428.89, -2.7, 184.96], [-0.121597, 0.696573, 0.706937, 0.015485], [0,0,0,0], [9E9, 9E9, 9E9, 9E9, 9E9, 9E9]];
	VAR robtarget OpenholeUD_6834 := [[432.84, -2.7, 184.34], [-0.109011, 0.698653, 0.707103, 0.002175], [0,0,0,0], [9E9, 9E9, 9E9, 9E9, 9E9, 9E9]];
	VAR robtarget OpenholeUD_6835 := [[436.79, -2.7, 183.72], [-0.096167, 0.700537, 0.707018, -0.011223], [0,0,0,0], [9E9, 9E9, 9E9, 9E9, 9E9, 9E9]];
	VAR robtarget OpenholeUD_6836 := [[440.75, -2.7, 183.09], [-0.083099, 0.702207, 0.706676, -0.024666], [0,0,0,0], [9E9, 9E9, 9E9, 9E9, 9E9, 9E9]];
	VAR robtarget OpenholeUD_6837 := [[444.7, -2.7, 182.47], [-0.069844, 0.703649, 0.706079, -0.038111], [0,0,0,0], [9E9, 9E9, 9E9, 9E9, 9E9, 9E9]];
	VAR robtarget OpenholeUD_6838 := [[448.65, -2.7, 181.85], [-0.056445, 0.70485, 0.705228, -0.051515], [0,0,0,0], [9E9, 9E9, 9E9, 9E9, 9E9, 9E9]];
	VAR robtarget OpenholeUD_6839 := [[452.6, -2.7, 181.23], [-0.042944, 0.705802, 0.704128, -0.064834], [0,0,0,0], [9E9, 9E9, 9E9, 9E9, 9E9, 9E9]];
	VAR robtarget OpenholeUD_6840 := [[456.55, -2.7, 180.61], [-0.029385, 0.706496, 0.702788, -0.078028], [0,0,0,0], [9E9, 9E9, 9E9, 9E9, 9E9, 9E9]];
	VAR robtarget OpenholeUD_6841 := [[460.5, -2.7, 179.99], [-0.015814, 0.70693, 0.70122, -0.091054], [0,0,0,0], [9E9, 9E9, 9E9, 9E9, 9E9, 9E9]];
	VAR robtarget OpenholeUD_6842 := [[464.45, -2.7, 179.37], [-0.002275, 0.707103, 0.699435, -0.103876], [0,0,0,0], [9E9, 9E9, 9E9, 9E9, 9E9, 9E9]];
